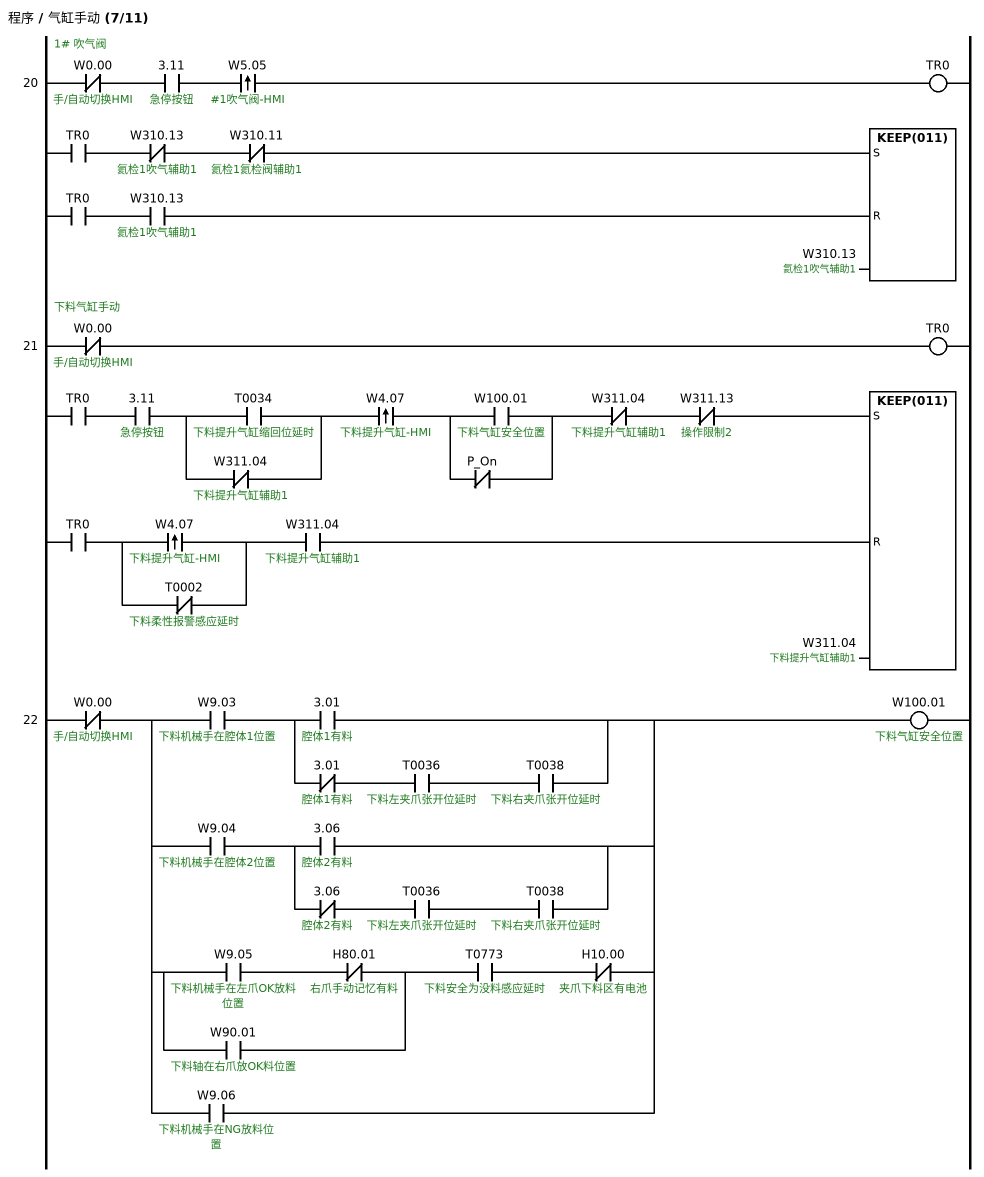
; [picture p120: 程序 / 气缸手动, rungs 20-22]
; rung 20: 1# 吹气阀
LDNOT W0.00  ; 手/自动切换HMI
AND 3.11  ; 急停按钮
@AND W5.05  ; #1吹气阀-HMI
OUT TR0
ANDNOT W310.13  ; 氦检1吹气辅助1
ANDNOT W310.11  ; 氦检1氦检阀辅助1
LD TR0
AND W310.13  ; 氦检1吹气辅助1
KEEP(011) W310.13  ; 氦检1吹气辅助1
; rung 21: 下料气缸手动
LDNOT W0.00  ; 手/自动切换HMI
OUT TR0
AND 3.11  ; 急停按钮
LD T0034  ; 下料提升气缸缩回位延时
ORNOT W311.04  ; 下料提升气缸辅助1
ANDLD
@AND W4.07  ; 下料提升气缸-HMI
LD W100.01  ; 下料气缸安全位置
ORNOT P_On
ANDLD
ANDNOT W311.04  ; 下料提升气缸辅助1
ANDNOT W311.13  ; 操作限制2
LD TR0
@LD W4.07  ; 下料提升气缸-HMI
ORNOT T0002  ; 下料柔性报警感应延时
ANDLD
AND W311.04  ; 下料提升气缸辅助1
KEEP(011) W311.04  ; 下料提升气缸辅助1
; rung 22
LDNOT W0.00  ; 手/自动切换HMI
LD W9.03  ; 下料机械手在腔体1位置
LD 3.01  ; 腔体1有料
LDNOT 3.01  ; 腔体1有料
AND T0036  ; 下料左夹爪张开位延时
AND T0038  ; 下料右夹爪张开位延时
ORLD
ANDLD
LD W9.04  ; 下料机械手在腔体2位置
LD 3.06  ; 腔体2有料
LDNOT 3.06  ; 腔体2有料
AND T0036  ; 下料左夹爪张开位延时
AND T0038  ; 下料右夹爪张开位延时
ORLD
ANDLD
ORLD
LD W9.05  ; 下料机械手在左爪OK放料位置
ANDNOT H80.01  ; 右爪手动记忆有料
OR W90.01  ; 下料轴在右爪放OK料位置
AND T0773  ; 下料安全为没料感应延时
ANDNOT H10.00  ; 夹爪下料区有电池
ORLD
OR W9.06  ; 下料机械手在NG放料位置
ANDLD
OUT W100.01  ; 下料气缸安全位置

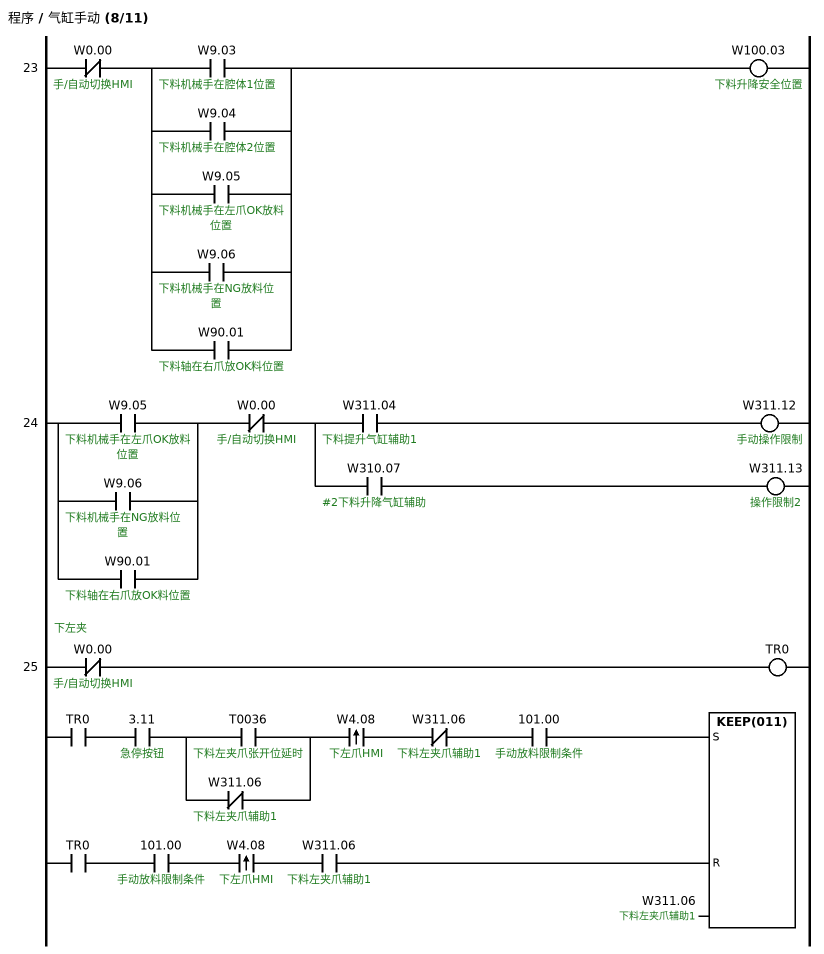
; rung 23
LDNOT W0.00  ; 手/自动切换HMI
LD W9.03  ; 下料机械手在腔体1位置
OR W9.04  ; 下料机械手在腔体2位置
OR W9.05  ; 下料机械手在左爪OK放料位置
OR W9.06  ; 下料机械手在NG放料位置
OR W90.01  ; 下料轴在右爪放OK料位置
ANDLD
OUT W100.03  ; 下料升降安全位置
; rung 24
LD W9.05  ; 下料机械手在左爪OK放料位置
OR W9.06  ; 下料机械手在NG放料位置
OR W90.01  ; 下料轴在右爪放OK料位置
ANDNOT W0.00  ; 手/自动切换HMI
OUT TR0
AND W311.04  ; 下料提升气缸辅助1
OUT W311.12  ; 手动操作限制
LD TR0
AND W310.07  ; #2下料升降气缸辅助
OUT W311.13  ; 操作限制2
; rung 25: 下左夹
LDNOT W0.00  ; 手/自动切换HMI
OUT TR0
AND 3.11  ; 急停按钮
LD T0036  ; 下料左夹爪张开位延时
ORNOT W311.06  ; 下料左夹爪辅助1
ANDLD
@AND W4.08  ; 下左爪HMI
ANDNOT W311.06  ; 下料左夹爪辅助1
AND 101.00  ; 手动放料限制条件
LD TR0
AND 101.00  ; 手动放料限制条件
@AND W4.08  ; 下左爪HMI
AND W311.06  ; 下料左夹爪辅助1
KEEP(011) W311.06  ; 下料左夹爪辅助1

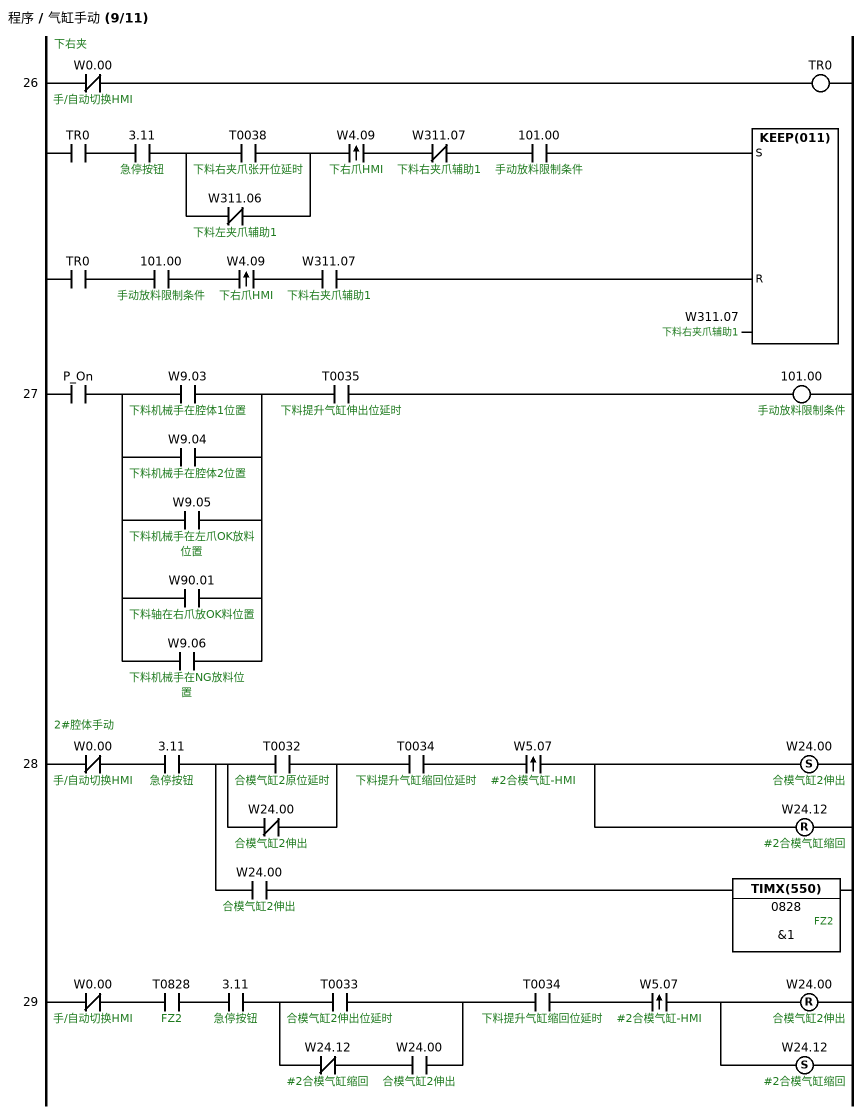
; rung 26: 下右夹
LDNOT W0.00  ; 手/自动切换HMI
OUT TR0
AND 3.11  ; 急停按钮
LD T0038  ; 下料右夹爪张开位延时
ORNOT W311.06  ; 下料左夹爪辅助1
ANDLD
@AND W4.09  ; 下右爪HMI
ANDNOT W311.07  ; 下料右夹爪辅助1
AND 101.00  ; 手动放料限制条件
LD TR0
AND 101.00  ; 手动放料限制条件
@AND W4.09  ; 下右爪HMI
AND W311.07  ; 下料右夹爪辅助1
KEEP(011) W311.07  ; 下料右夹爪辅助1
; rung 27
LD P_On
LD W9.03  ; 下料机械手在腔体1位置
OR W9.04  ; 下料机械手在腔体2位置
OR W9.05  ; 下料机械手在左爪OK放料位置
OR W90.01  ; 下料轴在右爪放OK料位置
OR W9.06  ; 下料机械手在NG放料位置
ANDLD
AND T0035  ; 下料提升气缸伸出位延时
OUT 101.00  ; 手动放料限制条件
; rung 28: 2#腔体手动
LDNOT W0.00  ; 手/自动切换HMI
AND 3.11  ; 急停按钮
OUT TR0
LD T0032  ; 合模气缸2原位延时
ORNOT W24.00  ; 合模气缸2伸出
ANDLD
AND T0034  ; 下料提升气缸缩回位延时
@AND W5.07  ; #2合模气缸-HMI
SET W24.00  ; 合模气缸2伸出
RSET W24.12  ; #2合模气缸缩回
LD TR0
AND W24.00  ; 合模气缸2伸出
TIMX(550) 0828 &1  ; FZ2
; rung 29
LDNOT W0.00  ; 手/自动切换HMI
AND T0828  ; FZ2
AND 3.11  ; 急停按钮
LD T0033  ; 合模气缸2伸出位延时
LDNOT W24.12  ; #2合模气缸缩回
AND W24.00  ; 合模气缸2伸出
ORLD
ANDLD
AND T0034  ; 下料提升气缸缩回位延时
@AND W5.07  ; #2合模气缸-HMI
RSET W24.00  ; 合模气缸2伸出
SET W24.12  ; #2合模气缸缩回

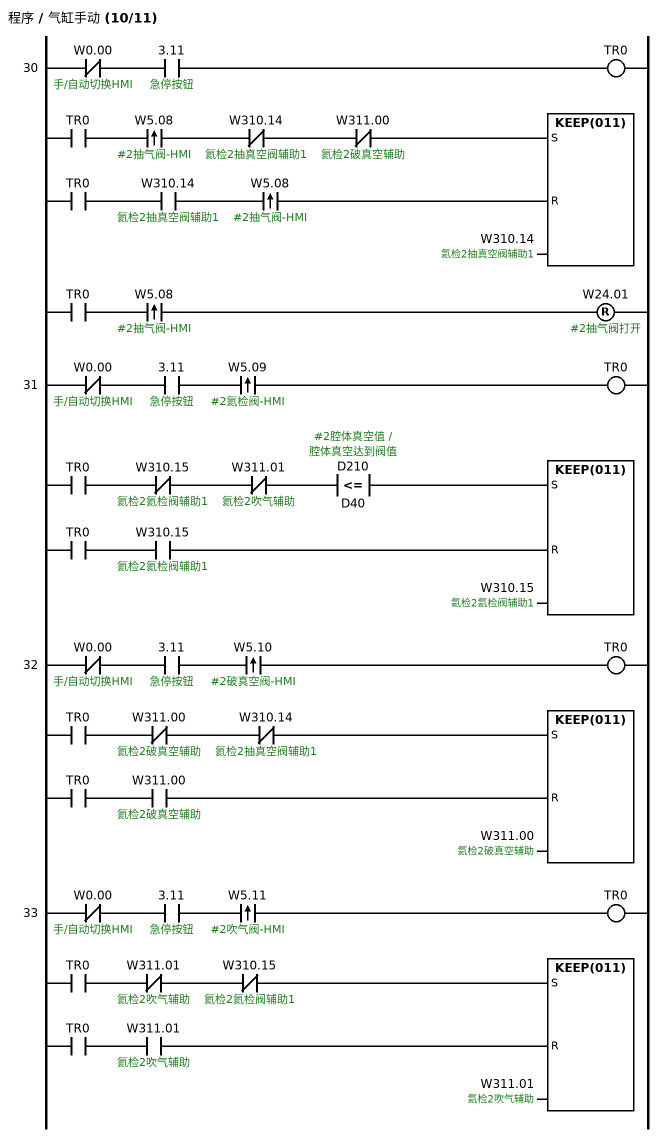
; rung 30
LDNOT W0.00  ; 手/自动切换HMI
AND 3.11  ; 急停按钮
OUT TR0
@AND W5.08  ; #2抽气阀-HMI
ANDNOT W310.14  ; 氦检2抽真空阀辅助1
ANDNOT W311.00  ; 氦检2破真空辅助
LD TR0
AND W310.14  ; 氦检2抽真空阀辅助1
@AND W5.08  ; #2抽气阀-HMI
KEEP(011) W310.14  ; 氦检2抽真空阀辅助1
LD TR0
@AND W5.08  ; #2抽气阀-HMI
RSET W24.01  ; #2抽气阀打开
; rung 31
LDNOT W0.00  ; 手/自动切换HMI
AND 3.11  ; 急停按钮
@AND W5.09  ; #2氦检阀-HMI
OUT TR0
ANDNOT W310.15  ; 氦检2氦检阀辅助1
ANDNOT W311.01  ; 氦检2吹气辅助
AND<=F(332) D210 D40  ; #2腔体真空值, 腔体真空达到阀值
LD TR0
AND W310.15  ; 氦检2氦检阀辅助1
KEEP(011) W310.15  ; 氦检2氦检阀辅助1
; rung 32
LDNOT W0.00  ; 手/自动切换HMI
AND 3.11  ; 急停按钮
@AND W5.10  ; #2破真空阀-HMI
OUT TR0
ANDNOT W311.00  ; 氦检2破真空辅助
ANDNOT W310.14  ; 氦检2抽真空阀辅助1
LD TR0
AND W311.00  ; 氦检2破真空辅助
KEEP(011) W311.00  ; 氦检2破真空辅助
; rung 33
LDNOT W0.00  ; 手/自动切换HMI
AND 3.11  ; 急停按钮
@AND W5.11  ; #2吹气阀-HMI
OUT TR0
ANDNOT W311.01  ; 氦检2吹气辅助
ANDNOT W310.15  ; 氦检2氦检阀辅助1
LD TR0
AND W311.01  ; 氦检2吹气辅助
KEEP(011) W311.01  ; 氦检2吹气辅助

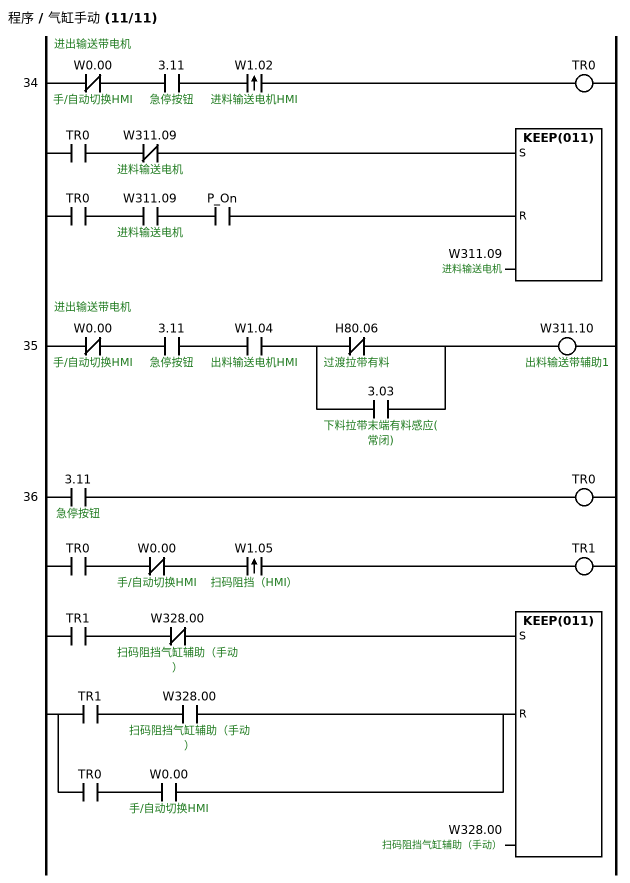
; rung 34: 进出输送带电机
LDNOT W0.00  ; 手/自动切换HMI
AND 3.11  ; 急停按钮
@AND W1.02  ; 进料输送电机HMI
OUT TR0
ANDNOT W311.09  ; 进料输送电机
LD TR0
AND W311.09  ; 进料输送电机
AND P_On
KEEP(011) W311.09  ; 进料输送电机
; rung 35: 进出输送带电机
LDNOT W0.00  ; 手/自动切换HMI
AND 3.11  ; 急停按钮
AND W1.04  ; 出料输送电机HMI
LDNOT H80.06  ; 过渡拉带有料
OR 3.03  ; 下料拉带末端有料感应(常闭)
ANDLD
OUT W311.10  ; 出料输送带辅助1
; rung 36
LD 3.11  ; 急停按钮
OUT TR0
ANDNOT W0.00  ; 手/自动切换HMI
@AND W1.05  ; 扫码阻挡（HMI）
OUT TR1
ANDNOT W328.00  ; 扫码阻挡气缸辅助（手动）
LD TR1
AND W328.00  ; 扫码阻挡气缸辅助（手动）
LD TR0
AND W0.00  ; 手/自动切换HMI
ORLD
KEEP(011) W328.00  ; 扫码阻挡气缸辅助（手动）

### Section 伺服参数

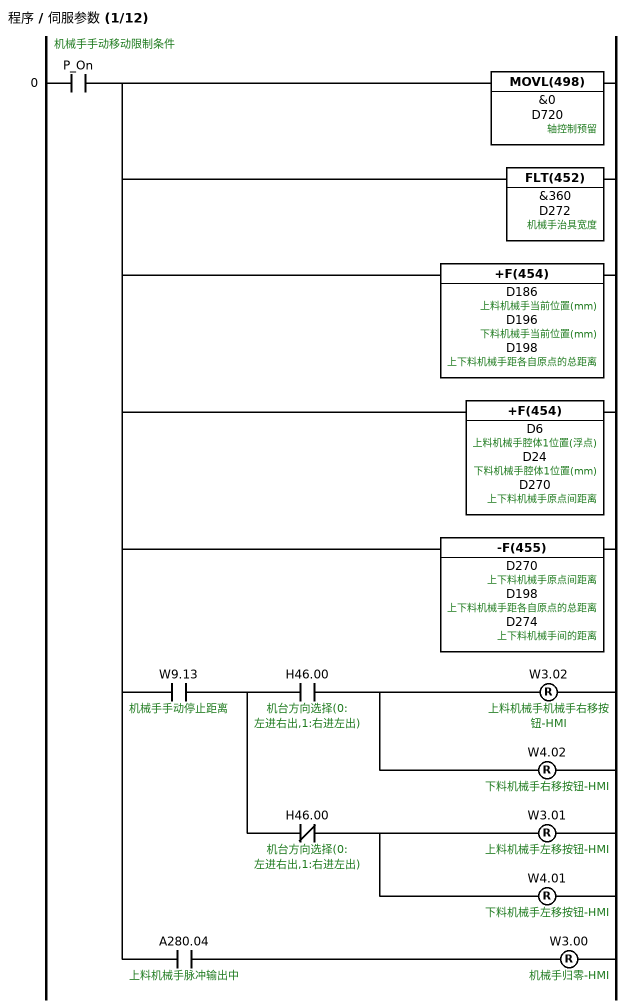
; rung 0: 机械手手动移动限制条件
LD P_On
OUT TR0
MOVL(498) &0 D720  ; 轴控制预留
FLT(452) &360 D272  ; 机械手治具宽度
+F(454) D186 D196 D198  ; 上料机械手当前位置(mm), 下料机械手当前位置(mm), 上下料机械手距各自原点的总距离
+F(454) D6 D24 D270  ; 上料机械手腔体1位置(浮点), 下料机械手腔体1位置(mm), 上下料机械手原点间距离
-F(455) D270 D198 D274  ; 上下料机械手原点间距离, 上下料机械手距各自原点的总距离, 上下料机械手间的距离
AND W9.13  ; 机械手手动停止距离
OUT TR1
AND H46.00  ; 机台方向选择(0:左进右出,1:右进左出)
RSET W3.02  ; 上料机械手机械手右移按钮-HMI
RSET W4.02  ; 下料机械手右移按钮-HMI
LD TR1
ANDNOT H46.00  ; 机台方向选择(0:左进右出,1:右进左出)
RSET W3.01  ; 上料机械手左移按钮-HMI
RSET W4.01  ; 下料机械手左移按钮-HMI
LD TR0
AND A280.04  ; 上料机械手脉冲输出中
RSET W3.00  ; 机械手归零-HMI

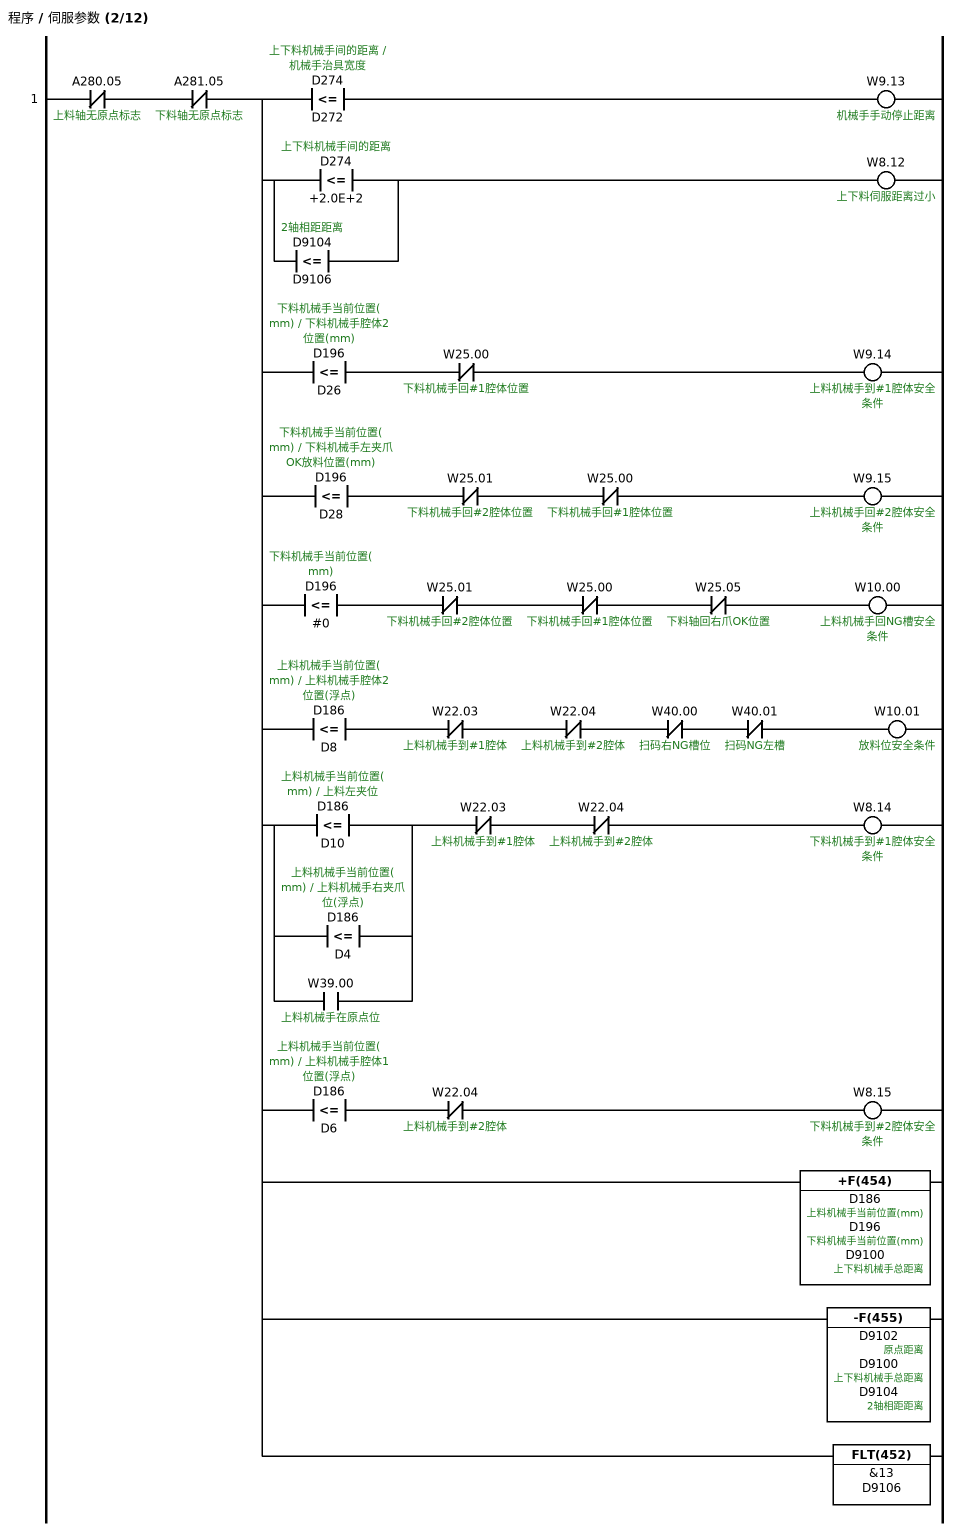
; rung 1
LDNOT A280.05  ; 上料轴无原点标志
ANDNOT A281.05  ; 下料轴无原点标志
OUT TR0
AND<=F(332) D274 D272  ; 上下料机械手间的距离, 机械手治具宽度
OUT W9.13  ; 机械手手动停止距离
LD TR0
LD<=F(332) D274 +2.0E+2  ; 上下料机械手间的距离
OR<=F(332) D9104 D9106  ; 2轴相距距离
ANDLD
OUT W8.12  ; 上下料伺服距离过小
LD TR0
AND<=F(332) D196 D26  ; 下料机械手当前位置(mm), 下料机械手腔体2位置(mm)
ANDNOT W25.00  ; 下料机械手回#1腔体位置
OUT W9.14  ; 上料机械手到#1腔体安全条件
LD TR0
AND<=F(332) D196 D28  ; 下料机械手当前位置(mm), 下料机械手左夹爪OK放料位置(mm)
ANDNOT W25.01  ; 下料机械手回#2腔体位置
ANDNOT W25.00  ; 下料机械手回#1腔体位置
OUT W9.15  ; 上料机械手回#2腔体安全条件
LD TR0
AND<=F(332) D196 #0  ; 下料机械手当前位置(mm)
ANDNOT W25.01  ; 下料机械手回#2腔体位置
ANDNOT W25.00  ; 下料机械手回#1腔体位置
ANDNOT W25.05  ; 下料轴回右爪OK位置
OUT W10.00  ; 上料机械手回NG槽安全条件
LD TR0
AND<=F(332) D186 D8  ; 上料机械手当前位置(mm), 上料机械手腔体2位置(浮点)
ANDNOT W22.03  ; 上料机械手到#1腔体
ANDNOT W22.04  ; 上料机械手到#2腔体
ANDNOT W40.00  ; 扫码右NG槽位
ANDNOT W40.01  ; 扫码NG左槽
OUT W10.01  ; 放料位安全条件
LD TR0
LD<=F(332) D186 D10  ; 上料机械手当前位置(mm), 上料左夹位
OR<=F(332) D186 D4  ; 上料机械手当前位置(mm), 上料机械手右夹爪位(浮点)
OR W39.00  ; 上料机械手在原点位
ANDLD
ANDNOT W22.03  ; 上料机械手到#1腔体
ANDNOT W22.04  ; 上料机械手到#2腔体
OUT W8.14  ; 下料机械手到#1腔体安全条件
LD TR0
AND<=F(332) D186 D6  ; 上料机械手当前位置(mm), 上料机械手腔体1位置(浮点)
ANDNOT W22.04  ; 上料机械手到#2腔体
OUT W8.15  ; 下料机械手到#2腔体安全条件
LD TR0
+F(454) D186 D196 D9100  ; 上料机械手当前位置(mm), 下料机械手当前位置(mm), 上下料机械手总距离
-F(455) D9102 D9100 D9104  ; 原点距离, 上下料机械手总距离, 2轴相距距离
FLT(452) &13 D9106

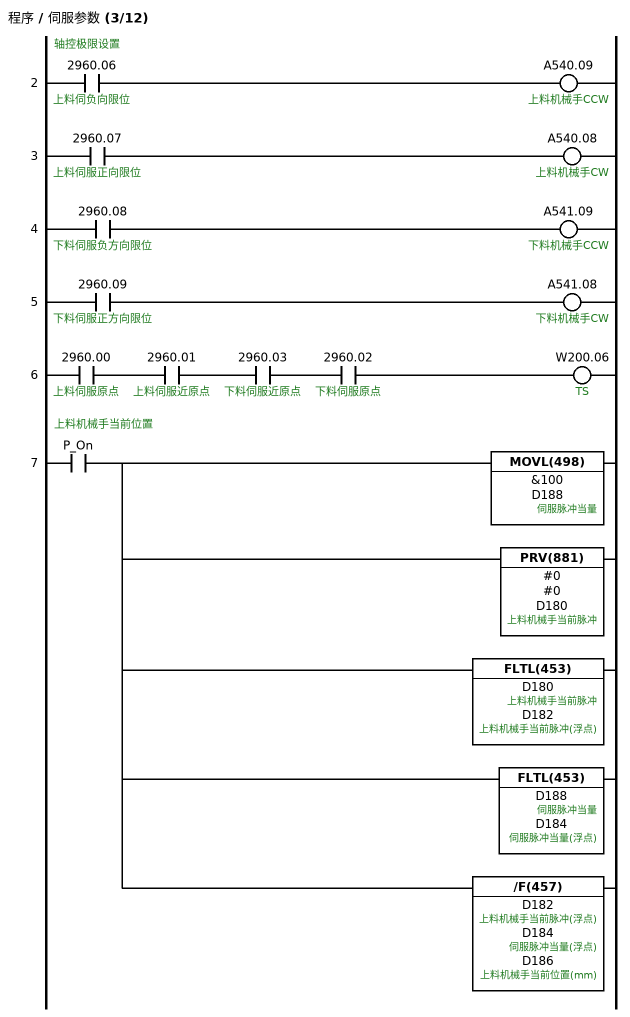
; rung 2: 轴控极限设置
LD 2960.06  ; 上料伺负向限位
OUT A540.09  ; 上料机械手CCW
; rung 3
LD 2960.07  ; 上料伺服正向限位
OUT A540.08  ; 上料机械手CW
; rung 4
LD 2960.08  ; 下料伺服负方向限位
OUT A541.09  ; 下料机械手CCW
; rung 5
LD 2960.09  ; 下料伺服正方向限位
OUT A541.08  ; 下料机械手CW
; rung 6
LD 2960.00  ; 上料伺服原点
AND 2960.01  ; 上料伺服近原点
AND 2960.03  ; 下料伺服近原点
AND 2960.02  ; 下料伺服原点
OUT W200.06  ; TS
; rung 7: 上料机械手当前位置
LD P_On
MOVL(498) &100 D188  ; 伺服脉冲当量
PRV(881) #0 #0 D180  ; 上料机械手当前脉冲
FLTL(453) D180 D182  ; 上料机械手当前脉冲, 上料机械手当前脉冲(浮点)
FLTL(453) D188 D184  ; 伺服脉冲当量, 伺服脉冲当量(浮点)
/F(457) D182 D184 D186  ; 上料机械手当前脉冲(浮点), 伺服脉冲当量(浮点), 上料机械手当前位置(mm)

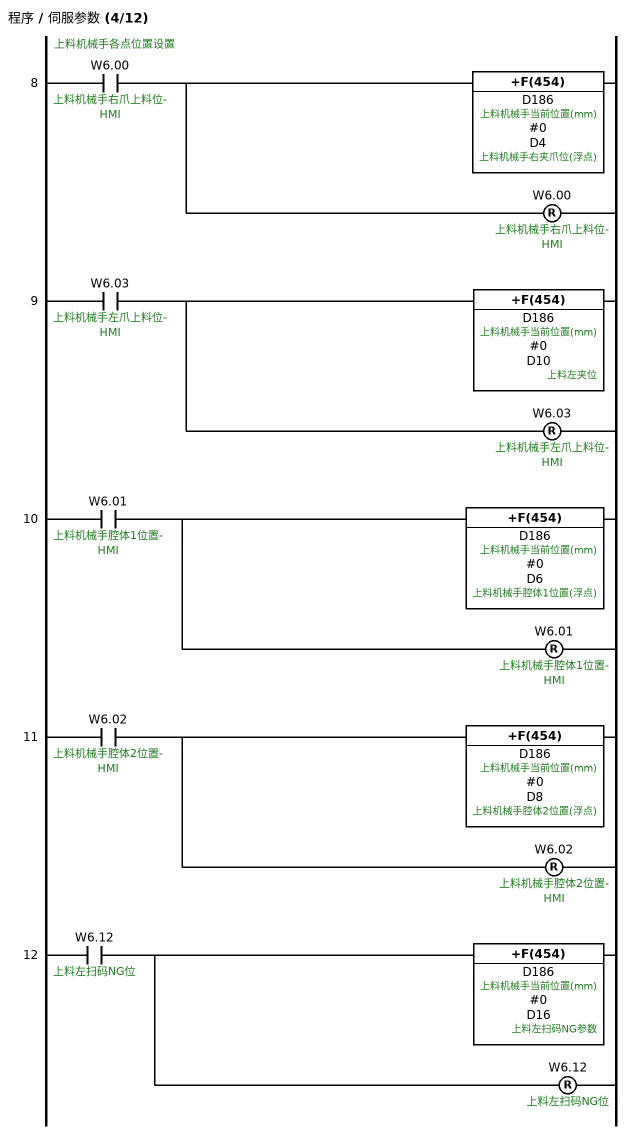
; rung 8: 上料机械手各点位置设置
LD W6.00  ; 上料机械手右爪上料位-HMI
+F(454) D186 #0 D4  ; 上料机械手当前位置(mm), 上料机械手右夹爪位(浮点)
RSET W6.00  ; 上料机械手右爪上料位-HMI
; rung 9
LD W6.03  ; 上料机械手左爪上料位-HMI
+F(454) D186 #0 D10  ; 上料机械手当前位置(mm), 上料左夹位
RSET W6.03  ; 上料机械手左爪上料位-HMI
; rung 10
LD W6.01  ; 上料机械手腔体1位置-HMI
+F(454) D186 #0 D6  ; 上料机械手当前位置(mm), 上料机械手腔体1位置(浮点)
RSET W6.01  ; 上料机械手腔体1位置-HMI
; rung 11
LD W6.02  ; 上料机械手腔体2位置-HMI
+F(454) D186 #0 D8  ; 上料机械手当前位置(mm), 上料机械手腔体2位置(浮点)
RSET W6.02  ; 上料机械手腔体2位置-HMI
; rung 12
LD W6.12  ; 上料左扫码NG位
+F(454) D186 #0 D16  ; 上料机械手当前位置(mm), 上料左扫码NG参数
RSET W6.12  ; 上料左扫码NG位

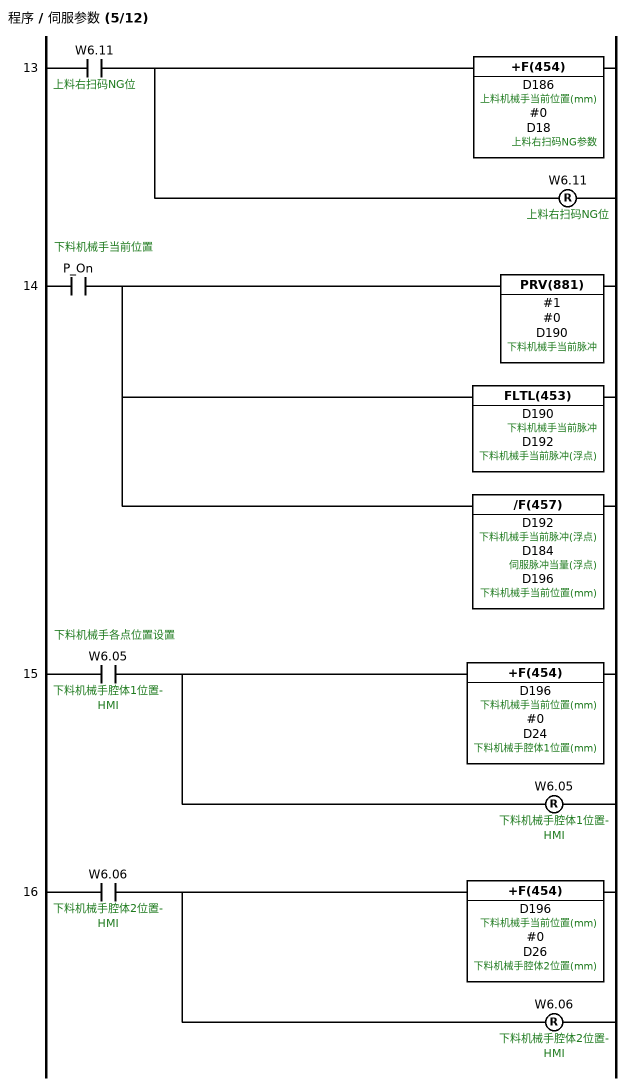
; rung 13
LD W6.11  ; 上料右扫码NG位
+F(454) D186 #0 D18  ; 上料机械手当前位置(mm), 上料右扫码NG参数
RSET W6.11  ; 上料右扫码NG位
; rung 14: 下料机械手当前位置
LD P_On
PRV(881) #1 #0 D190  ; 下料机械手当前脉冲
FLTL(453) D190 D192  ; 下料机械手当前脉冲, 下料机械手当前脉冲(浮点)
/F(457) D192 D184 D196  ; 下料机械手当前脉冲(浮点), 伺服脉冲当量(浮点), 下料机械手当前位置(mm)
; rung 15: 下料机械手各点位置设置
LD W6.05  ; 下料机械手腔体1位置-HMI
+F(454) D196 #0 D24  ; 下料机械手当前位置(mm), 下料机械手腔体1位置(mm)
RSET W6.05  ; 下料机械手腔体1位置-HMI
; rung 16
LD W6.06  ; 下料机械手腔体2位置-HMI
+F(454) D196 #0 D26  ; 下料机械手当前位置(mm), 下料机械手腔体2位置(mm)
RSET W6.06  ; 下料机械手腔体2位置-HMI

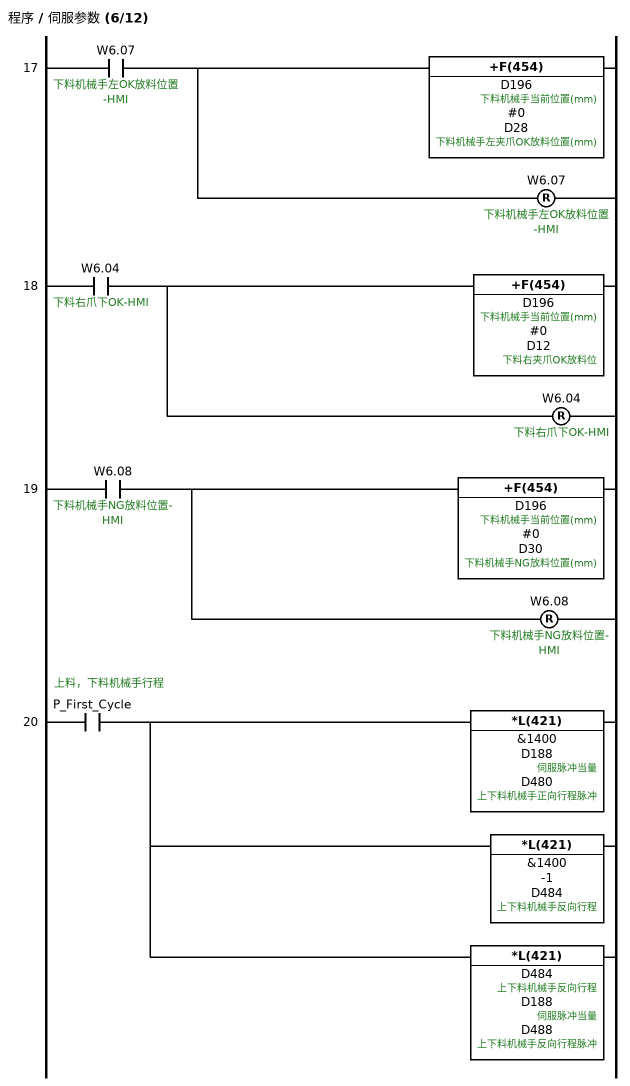
; rung 17
LD W6.07  ; 下料机械手左OK放料位置-HMI
+F(454) D196 #0 D28  ; 下料机械手当前位置(mm), 下料机械手左夹爪OK放料位置(mm)
RSET W6.07  ; 下料机械手左OK放料位置-HMI
; rung 18
LD W6.04  ; 下料右爪下OK-HMI
+F(454) D196 #0 D12  ; 下料机械手当前位置(mm), 下料右夹爪OK放料位
RSET W6.04  ; 下料右爪下OK-HMI
; rung 19
LD W6.08  ; 下料机械手NG放料位置-HMI
+F(454) D196 #0 D30  ; 下料机械手当前位置(mm), 下料机械手NG放料位置(mm)
RSET W6.08  ; 下料机械手NG放料位置-HMI
; rung 20: 上料，下料机械手行程
LD P_First_Cycle
*L(421) &1400 D188 D480  ; 伺服脉冲当量, 上下料机械手正向行程脉冲
*L(421) &1400 -1 D484  ; 上下料机械手反向行程
*L(421) D484 D188 D488  ; 上下料机械手反向行程, 伺服脉冲当量, 上下料机械手反向行程脉冲

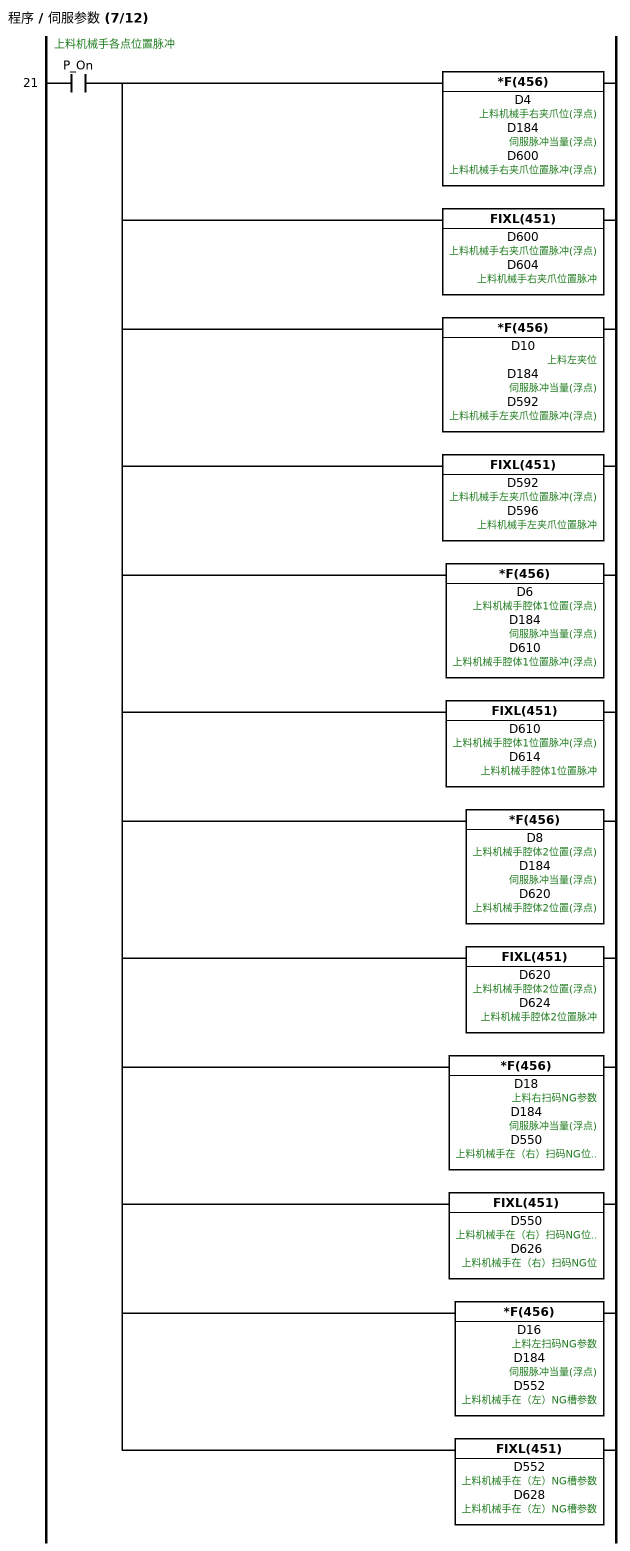
; rung 21: 上料机械手各点位置脉冲
LD P_On
*F(456) D4 D184 D600  ; 上料机械手右夹爪位(浮点), 伺服脉冲当量(浮点), 上料机械手右夹爪位置脉冲(浮点)
FIXL(451) D600 D604  ; 上料机械手右夹爪位置脉冲(浮点), 上料机械手右夹爪位置脉冲
*F(456) D10 D184 D592  ; 上料左夹位, 伺服脉冲当量(浮点), 上料机械手左夹爪位置脉冲(浮点)
FIXL(451) D592 D596  ; 上料机械手左夹爪位置脉冲(浮点), 上料机械手左夹爪位置脉冲
*F(456) D6 D184 D610  ; 上料机械手腔体1位置(浮点), 伺服脉冲当量(浮点), 上料机械手腔体1位置脉冲(浮点)
FIXL(451) D610 D614  ; 上料机械手腔体1位置脉冲(浮点), 上料机械手腔体1位置脉冲
*F(456) D8 D184 D620  ; 上料机械手腔体2位置(浮点), 伺服脉冲当量(浮点)
FIXL(451) D620 D624  ; 上料机械手腔体2位置(浮点), 上料机械手腔体2位置脉冲
*F(456) D18 D184 D550  ; 上料右扫码NG参数, 伺服脉冲当量(浮点), 上料机械手在（右）扫码NG位..
FIXL(451) D550 D626  ; 上料机械手在（右）扫码NG位.., 上料机械手在（右）扫码NG位
*F(456) D16 D184 D552  ; 上料左扫码NG参数, 伺服脉冲当量(浮点), 上料机械手在（左）NG槽参数
FIXL(451) D552 D628  ; 上料机械手在（左）NG槽参数

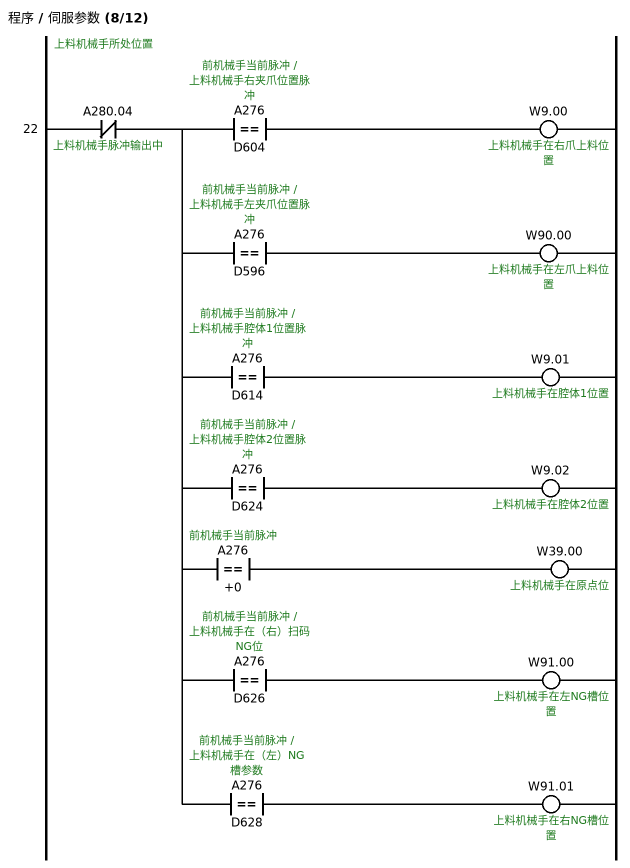
; rung 22: 上料机械手所处位置
LDNOT A280.04  ; 上料机械手脉冲输出中
OUT TR0
AND=SL(303) A276 D604  ; 前机械手当前脉冲, 上料机械手右夹爪位置脉冲
OUT W9.00  ; 上料机械手在右爪上料位置
LD TR0
AND=SL(303) A276 D596  ; 前机械手当前脉冲, 上料机械手左夹爪位置脉冲
OUT W90.00  ; 上料机械手在左爪上料位置
LD TR0
AND=SL(303) A276 D614  ; 前机械手当前脉冲, 上料机械手腔体1位置脉冲
OUT W9.01  ; 上料机械手在腔体1位置
LD TR0
AND=SL(303) A276 D624  ; 前机械手当前脉冲, 上料机械手腔体2位置脉冲
OUT W9.02  ; 上料机械手在腔体2位置
LD TR0
AND=SL(303) A276 +0  ; 前机械手当前脉冲
OUT W39.00  ; 上料机械手在原点位
LD TR0
AND=SL(303) A276 D626  ; 前机械手当前脉冲, 上料机械手在（右）扫码NG位
OUT W91.00  ; 上料机械手在左NG槽位置
LD TR0
AND=SL(303) A276 D628  ; 前机械手当前脉冲, 上料机械手在（左）NG槽参数
OUT W91.01  ; 上料机械手在右NG槽位置

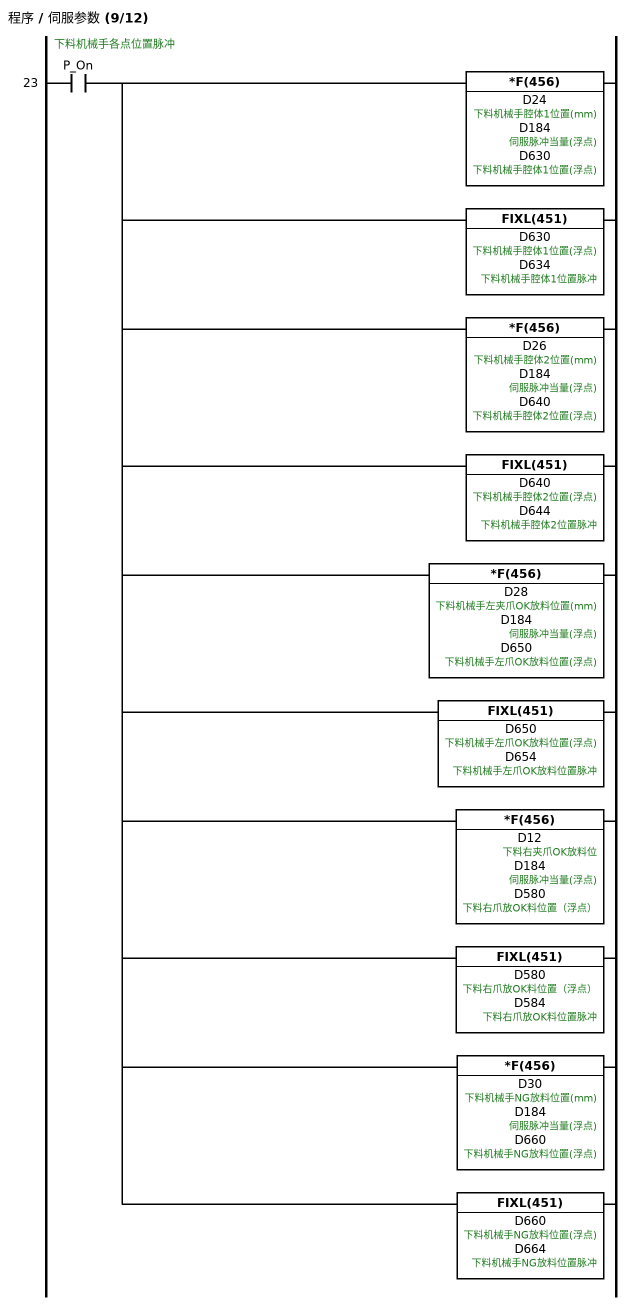
; rung 23: 下料机械手各点位置脉冲
LD P_On
*F(456) D24 D184 D630  ; 下料机械手腔体1位置(mm), 伺服脉冲当量(浮点), 下料机械手腔体1位置(浮点)
FIXL(451) D630 D634  ; 下料机械手腔体1位置(浮点), 下料机械手腔体1位置脉冲
*F(456) D26 D184 D640  ; 下料机械手腔体2位置(mm), 伺服脉冲当量(浮点), 下料机械手腔体2位置(浮点)
FIXL(451) D640 D644  ; 下料机械手腔体2位置(浮点), 下料机械手腔体2位置脉冲
*F(456) D28 D184 D650  ; 下料机械手左夹爪OK放料位置(mm), 伺服脉冲当量(浮点), 下料机械手左爪OK放料位置(浮点)
FIXL(451) D650 D654  ; 下料机械手左爪OK放料位置(浮点), 下料机械手左爪OK放料位置脉冲
*F(456) D12 D184 D580  ; 下料右夹爪OK放料位, 伺服脉冲当量(浮点), 下料右爪放OK料位置（浮点）
FIXL(451) D580 D584  ; 下料右爪放OK料位置（浮点）, 下料右爪放OK料位置脉冲
*F(456) D30 D184 D660  ; 下料机械手NG放料位置(mm), 伺服脉冲当量(浮点), 下料机械手NG放料位置(浮点)
FIXL(451) D660 D664  ; 下料机械手NG放料位置(浮点), 下料机械手NG放料位置脉冲

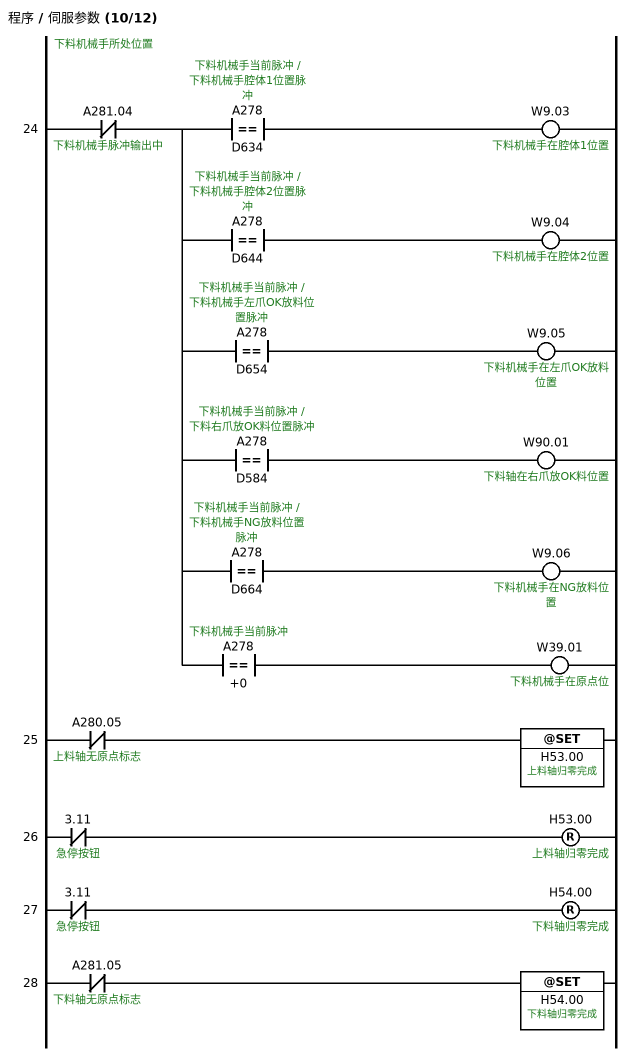
; rung 24: 下料机械手所处位置
LDNOT A281.04  ; 下料机械手脉冲输出中
OUT TR0
AND=SL(303) A278 D634  ; 下料机械手当前脉冲, 下料机械手腔体1位置脉冲
OUT W9.03  ; 下料机械手在腔体1位置
LD TR0
AND=SL(303) A278 D644  ; 下料机械手当前脉冲, 下料机械手腔体2位置脉冲
OUT W9.04  ; 下料机械手在腔体2位置
LD TR0
AND=SL(303) A278 D654  ; 下料机械手当前脉冲, 下料机械手左爪OK放料位置脉冲
OUT W9.05  ; 下料机械手在左爪OK放料位置
LD TR0
AND=SL(303) A278 D584  ; 下料机械手当前脉冲, 下料右爪放OK料位置脉冲
OUT W90.01  ; 下料轴在右爪放OK料位置
LD TR0
AND=SL(303) A278 D664  ; 下料机械手当前脉冲, 下料机械手NG放料位置脉冲
OUT W9.06  ; 下料机械手在NG放料位置
LD TR0
AND=SL(303) A278 +0  ; 下料机械手当前脉冲
OUT W39.01  ; 下料机械手在原点位
; rung 25
LDNOT A280.05  ; 上料轴无原点标志
@SET H53.00  ; 上料轴归零完成
; rung 26
LDNOT 3.11  ; 急停按钮
RSET H53.00  ; 上料轴归零完成
; rung 27
LDNOT 3.11  ; 急停按钮
RSET H54.00  ; 下料轴归零完成
; rung 28
LDNOT A281.05  ; 下料轴无原点标志
@SET H54.00  ; 下料轴归零完成

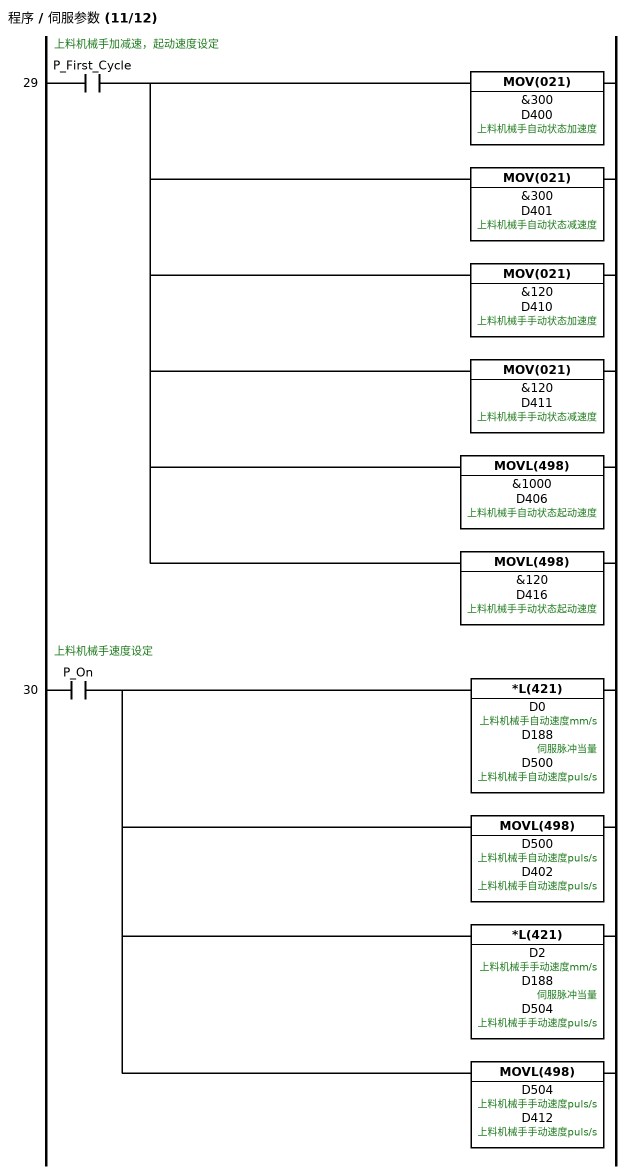
; rung 29: 上料机械手加减速，起动速度设定
LD P_First_Cycle
MOV(021) &300 D400  ; 上料机械手自动状态加速度
MOV(021) &300 D401  ; 上料机械手自动状态减速度
MOV(021) &120 D410  ; 上料机械手手动状态加速度
MOV(021) &120 D411  ; 上料机械手手动状态减速度
MOVL(498) &1000 D406  ; 上料机械手自动状态起动速度
MOVL(498) &120 D416  ; 上料机械手手动状态起动速度
; rung 30: 上料机械手速度设定
LD P_On
*L(421) D0 D188 D500  ; 上料机械手自动速度mm/s, 伺服脉冲当量, 上料机械手自动速度puls/s
MOVL(498) D500 D402  ; 上料机械手自动速度puls/s
*L(421) D2 D188 D504  ; 上料机械手手动速度mm/s, 伺服脉冲当量, 上料机械手手动速度puls/s
MOVL(498) D504 D412  ; 上料机械手手动速度puls/s

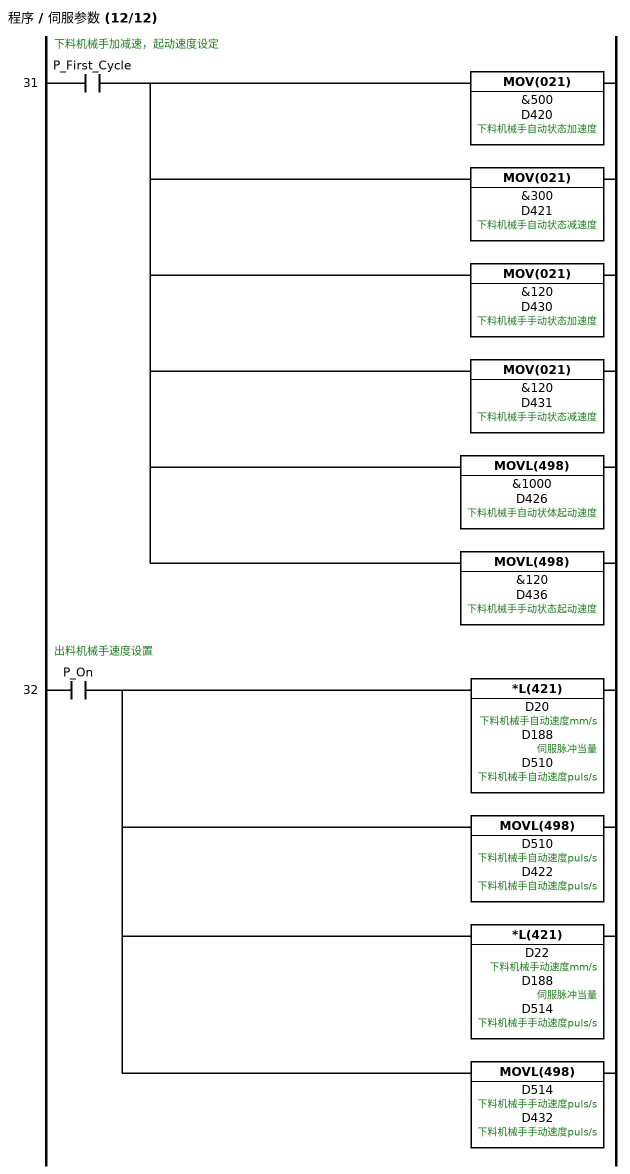
; rung 31: 下料机械手加减速，起动速度设定
LD P_First_Cycle
MOV(021) &500 D420  ; 下料机械手自动状态加速度
MOV(021) &300 D421  ; 下料机械手自动状态减速度
MOV(021) &120 D430  ; 下料机械手手动状态加速度
MOV(021) &120 D431  ; 下料机械手手动状态减速度
MOVL(498) &1000 D426  ; 下料机械手自动状体起动速度
MOVL(498) &120 D436  ; 下料机械手手动状态起动速度
; rung 32: 出料机械手速度设置
LD P_On
*L(421) D20 D188 D510  ; 下料机械手自动速度mm/s, 伺服脉冲当量, 下料机械手自动速度puls/s
MOVL(498) D510 D422  ; 下料机械手自动速度puls/s
*L(421) D22 D188 D514  ; 下料机械手动速度mm/s, 伺服脉冲当量, 下料机械手手动速度puls/s
MOVL(498) D514 D432  ; 下料机械手手动速度puls/s

### Section 伺服手动

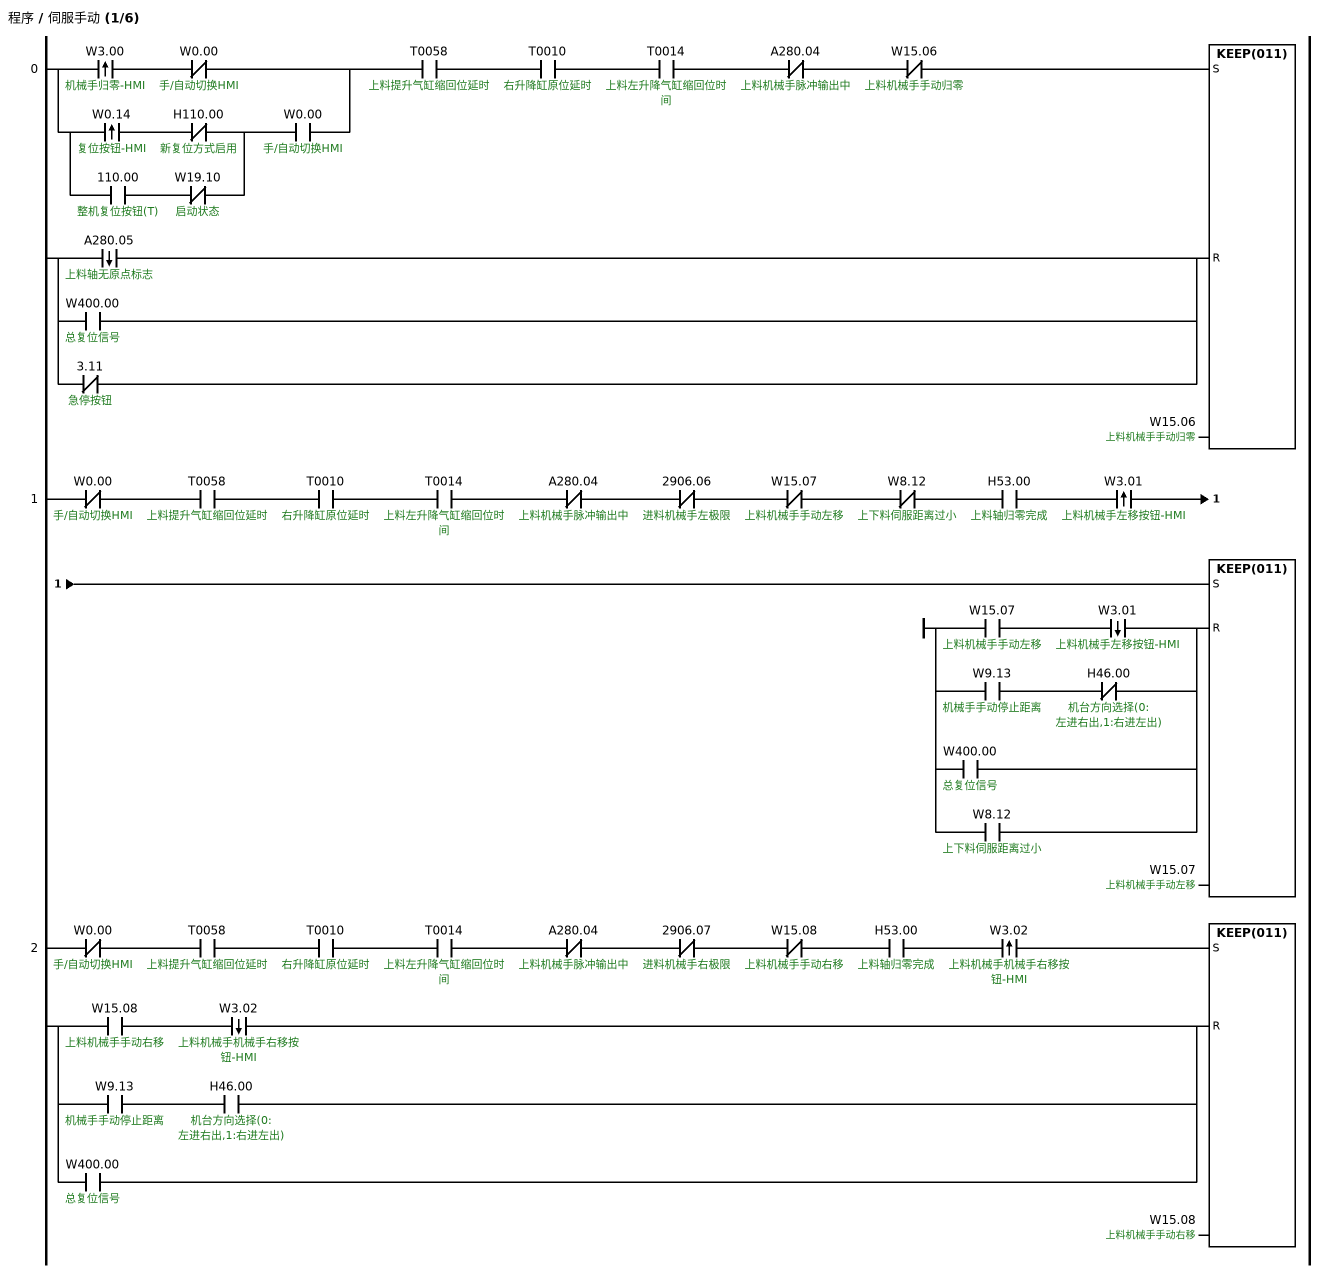
; rung 0
@LD W3.00  ; 机械手归零-HMI
ANDNOT W0.00  ; 手/自动切换HMI
@LD W0.14  ; 复位按钮-HMI
ANDNOT H110.00  ; 新复位方式启用
LD 110.00  ; 整机复位按钮(T)
ANDNOT W19.10  ; 启动状态
ORLD
AND W0.00  ; 手/自动切换HMI
ORLD
AND T0058  ; 上料提升气缸缩回位延时
AND T0010  ; 右升降缸原位延时
AND T0014  ; 上料左升降气缸缩回位时间
ANDNOT A280.04  ; 上料机械手脉冲输出中
ANDNOT W15.06  ; 上料机械手手动归零
%LD A280.05  ; 上料轴无原点标志
OR W400.00  ; 总复位信号
ORNOT 3.11  ; 急停按钮
KEEP(011) W15.06  ; 上料机械手手动归零
; rung 1
LDNOT W0.00  ; 手/自动切换HMI
AND T0058  ; 上料提升气缸缩回位延时
AND T0010  ; 右升降缸原位延时
AND T0014  ; 上料左升降气缸缩回位时间
ANDNOT A280.04  ; 上料机械手脉冲输出中
ANDNOT 2906.06  ; 进料机械手左极限
ANDNOT W15.07  ; 上料机械手手动左移
ANDNOT W8.12  ; 上下料伺服距离过小
AND H53.00  ; 上料轴归零完成
@AND W3.01  ; 上料机械手左移按钮-HMI
LD W15.07  ; 上料机械手手动左移
%AND W3.01  ; 上料机械手左移按钮-HMI
LD W9.13  ; 机械手手动停止距离
ANDNOT H46.00  ; 机台方向选择(0:左进右出,1:右进左出)
ORLD
OR W400.00  ; 总复位信号
OR W8.12  ; 上下料伺服距离过小
KEEP(011) W15.07  ; 上料机械手手动左移
; rung 2
LDNOT W0.00  ; 手/自动切换HMI
AND T0058  ; 上料提升气缸缩回位延时
AND T0010  ; 右升降缸原位延时
AND T0014  ; 上料左升降气缸缩回位时间
ANDNOT A280.04  ; 上料机械手脉冲输出中
ANDNOT 2906.07  ; 进料机械手右极限
ANDNOT W15.08  ; 上料机械手手动右移
AND H53.00  ; 上料轴归零完成
@AND W3.02  ; 上料机械手机械手右移按钮-HMI
LD W15.08  ; 上料机械手手动右移
%AND W3.02  ; 上料机械手机械手右移按钮-HMI
LD W9.13  ; 机械手手动停止距离
AND H46.00  ; 机台方向选择(0:左进右出,1:右进左出)
ORLD
OR W400.00  ; 总复位信号
KEEP(011) W15.08  ; 上料机械手手动右移

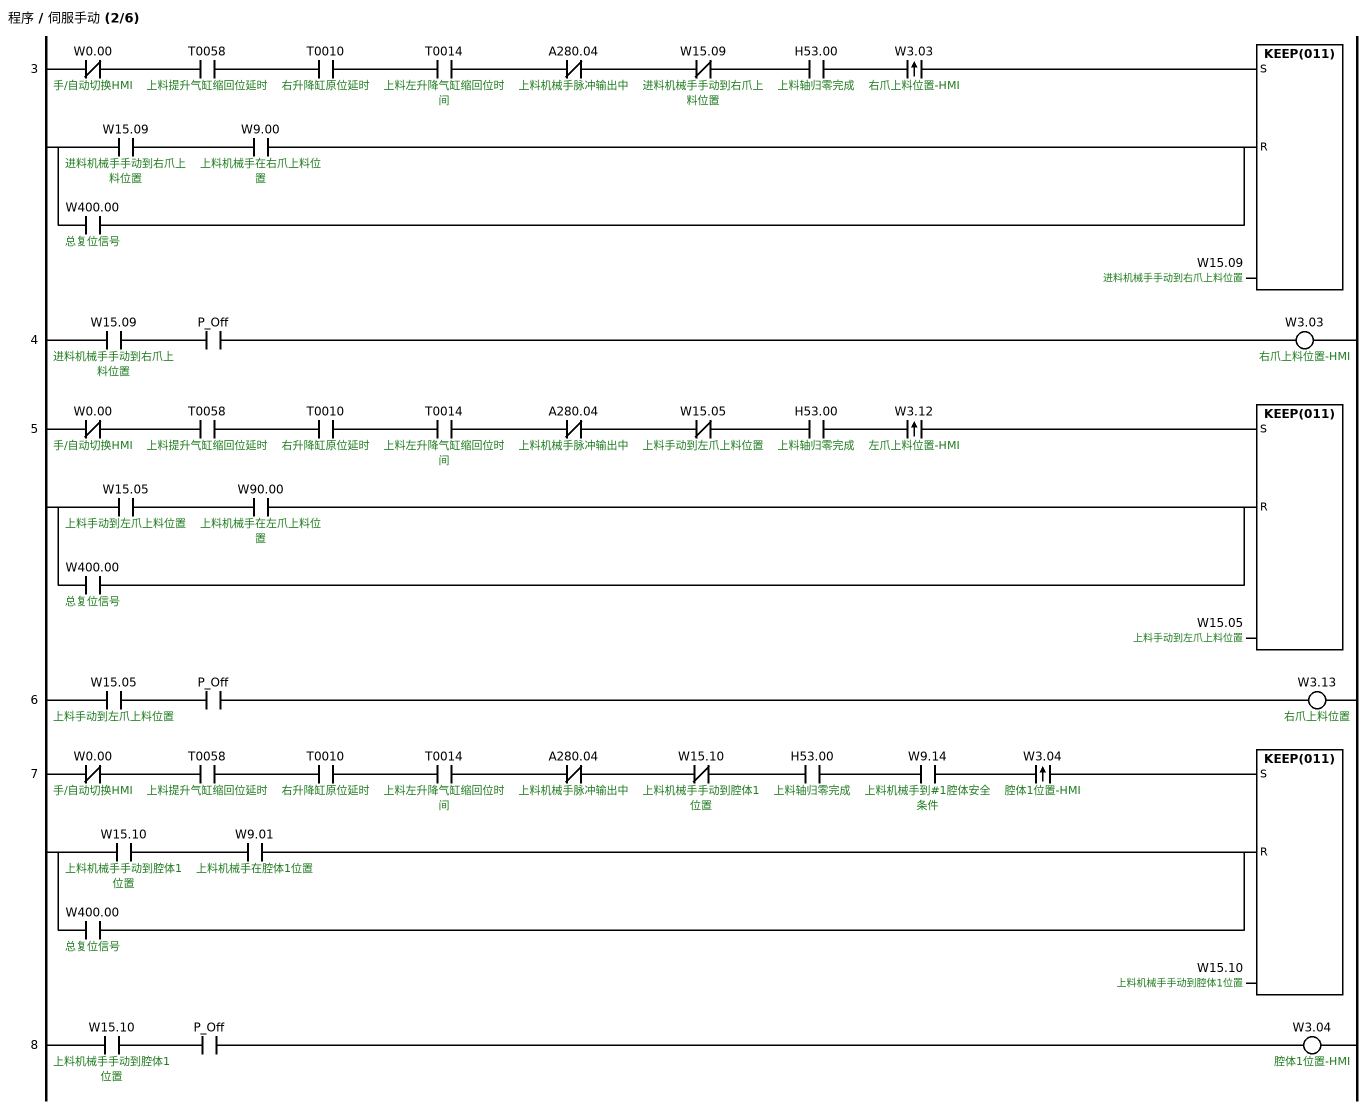
; rung 3
LDNOT W0.00  ; 手/自动切换HMI
AND T0058  ; 上料提升气缸缩回位延时
AND T0010  ; 右升降缸原位延时
AND T0014  ; 上料左升降气缸缩回位时间
ANDNOT A280.04  ; 上料机械手脉冲输出中
ANDNOT W15.09  ; 进料机械手手动到右爪上料位置
AND H53.00  ; 上料轴归零完成
@AND W3.03  ; 右爪上料位置-HMI
LD W15.09  ; 进料机械手手动到右爪上料位置
AND W9.00  ; 上料机械手在右爪上料位置
OR W400.00  ; 总复位信号
KEEP(011) W15.09  ; 进料机械手手动到右爪上料位置
; rung 4
LD W15.09  ; 进料机械手手动到右爪上料位置
AND P_Off
OUT W3.03  ; 右爪上料位置-HMI
; rung 5
LDNOT W0.00  ; 手/自动切换HMI
AND T0058  ; 上料提升气缸缩回位延时
AND T0010  ; 右升降缸原位延时
AND T0014  ; 上料左升降气缸缩回位时间
ANDNOT A280.04  ; 上料机械手脉冲输出中
ANDNOT W15.05  ; 上料手动到左爪上料位置
AND H53.00  ; 上料轴归零完成
@AND W3.12  ; 左爪上料位置-HMI
LD W15.05  ; 上料手动到左爪上料位置
AND W90.00  ; 上料机械手在左爪上料位置
OR W400.00  ; 总复位信号
KEEP(011) W15.05  ; 上料手动到左爪上料位置
; rung 6
LD W15.05  ; 上料手动到左爪上料位置
AND P_Off
OUT W3.13  ; 右爪上料位置
; rung 7
LDNOT W0.00  ; 手/自动切换HMI
AND T0058  ; 上料提升气缸缩回位延时
AND T0010  ; 右升降缸原位延时
AND T0014  ; 上料左升降气缸缩回位时间
ANDNOT A280.04  ; 上料机械手脉冲输出中
ANDNOT W15.10  ; 上料机械手手动到腔体1位置
AND H53.00  ; 上料轴归零完成
AND W9.14  ; 上料机械手到#1腔体安全条件
@AND W3.04  ; 腔体1位置-HMI
LD W15.10  ; 上料机械手手动到腔体1位置
AND W9.01  ; 上料机械手在腔体1位置
OR W400.00  ; 总复位信号
KEEP(011) W15.10  ; 上料机械手手动到腔体1位置
; rung 8
LD W15.10  ; 上料机械手手动到腔体1位置
AND P_Off
OUT W3.04  ; 腔体1位置-HMI

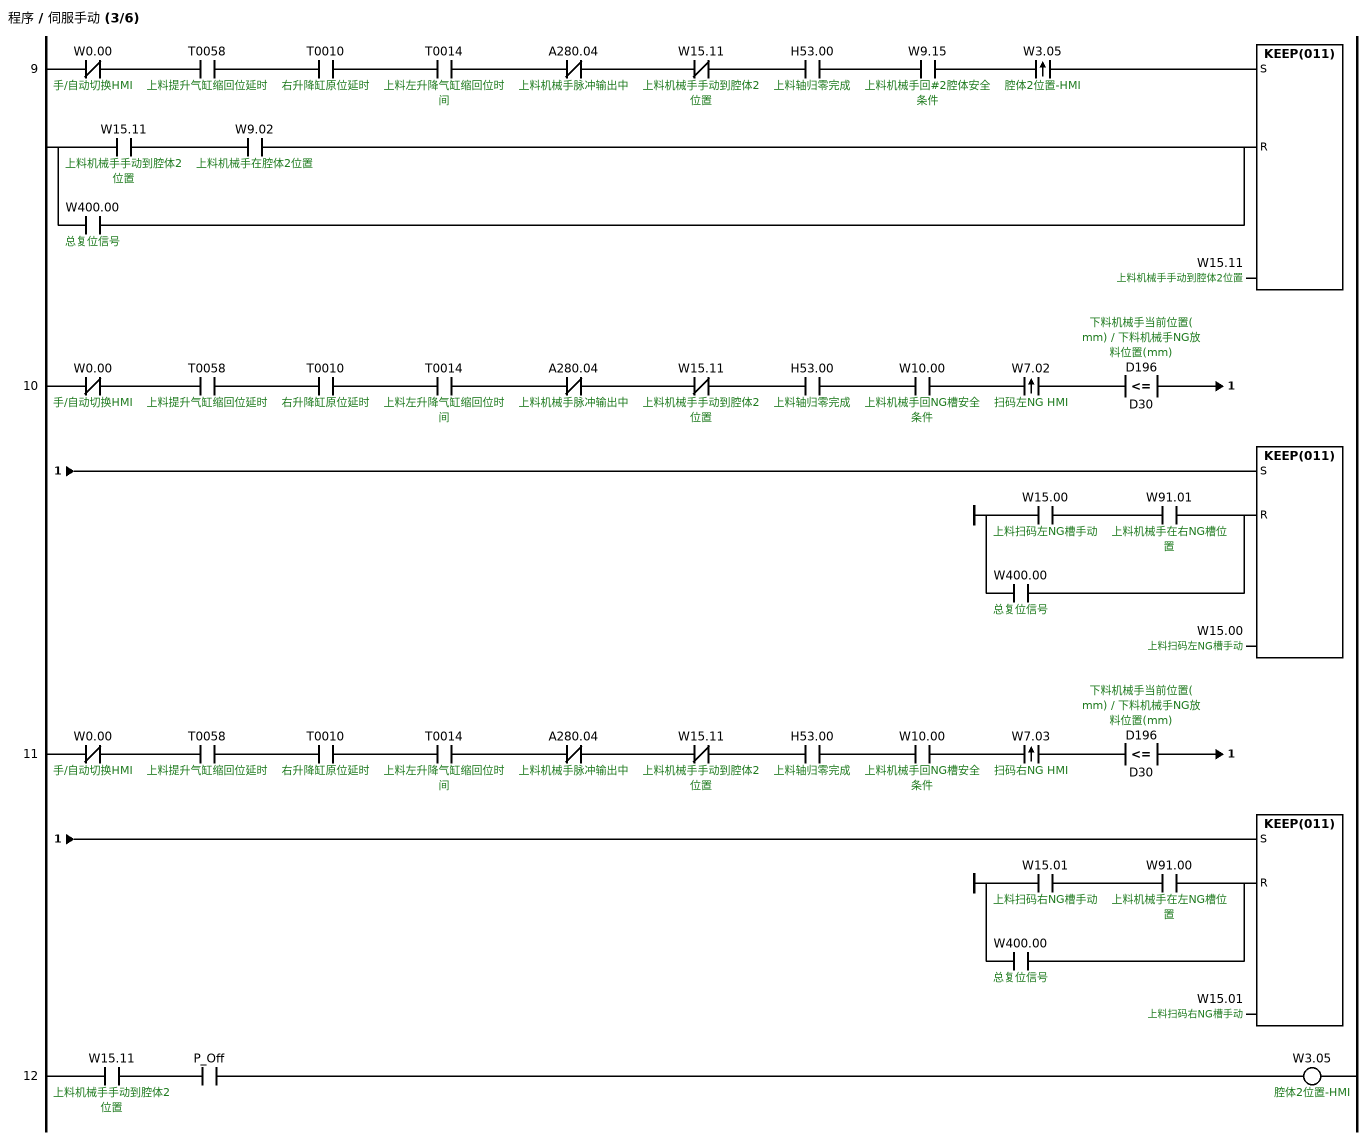
; rung 9
LDNOT W0.00  ; 手/自动切换HMI
AND T0058  ; 上料提升气缸缩回位延时
AND T0010  ; 右升降缸原位延时
AND T0014  ; 上料左升降气缸缩回位时间
ANDNOT A280.04  ; 上料机械手脉冲输出中
ANDNOT W15.11  ; 上料机械手手动到腔体2位置
AND H53.00  ; 上料轴归零完成
AND W9.15  ; 上料机械手回#2腔体安全条件
@AND W3.05  ; 腔体2位置-HMI
LD W15.11  ; 上料机械手手动到腔体2位置
AND W9.02  ; 上料机械手在腔体2位置
OR W400.00  ; 总复位信号
KEEP(011) W15.11  ; 上料机械手手动到腔体2位置
; rung 10
LDNOT W0.00  ; 手/自动切换HMI
AND T0058  ; 上料提升气缸缩回位延时
AND T0010  ; 右升降缸原位延时
AND T0014  ; 上料左升降气缸缩回位时间
ANDNOT A280.04  ; 上料机械手脉冲输出中
ANDNOT W15.11  ; 上料机械手手动到腔体2位置
AND H53.00  ; 上料轴归零完成
AND W10.00  ; 上料机械手回NG槽安全条件
@AND W7.02  ; 扫码左NG HMI
AND<=F(332) D196 D30  ; 下料机械手当前位置(mm), 下料机械手NG放料位置(mm)
LD W15.00  ; 上料扫码左NG槽手动
AND W91.01  ; 上料机械手在右NG槽位置
OR W400.00  ; 总复位信号
KEEP(011) W15.00  ; 上料扫码左NG槽手动
; rung 11
LDNOT W0.00  ; 手/自动切换HMI
AND T0058  ; 上料提升气缸缩回位延时
AND T0010  ; 右升降缸原位延时
AND T0014  ; 上料左升降气缸缩回位时间
ANDNOT A280.04  ; 上料机械手脉冲输出中
ANDNOT W15.11  ; 上料机械手手动到腔体2位置
AND H53.00  ; 上料轴归零完成
AND W10.00  ; 上料机械手回NG槽安全条件
@AND W7.03  ; 扫码右NG HMI
AND<=F(332) D196 D30  ; 下料机械手当前位置(mm), 下料机械手NG放料位置(mm)
LD W15.01  ; 上料扫码右NG槽手动
AND W91.00  ; 上料机械手在左NG槽位置
OR W400.00  ; 总复位信号
KEEP(011) W15.01  ; 上料扫码右NG槽手动
; rung 12
LD W15.11  ; 上料机械手手动到腔体2位置
AND P_Off
OUT W3.05  ; 腔体2位置-HMI

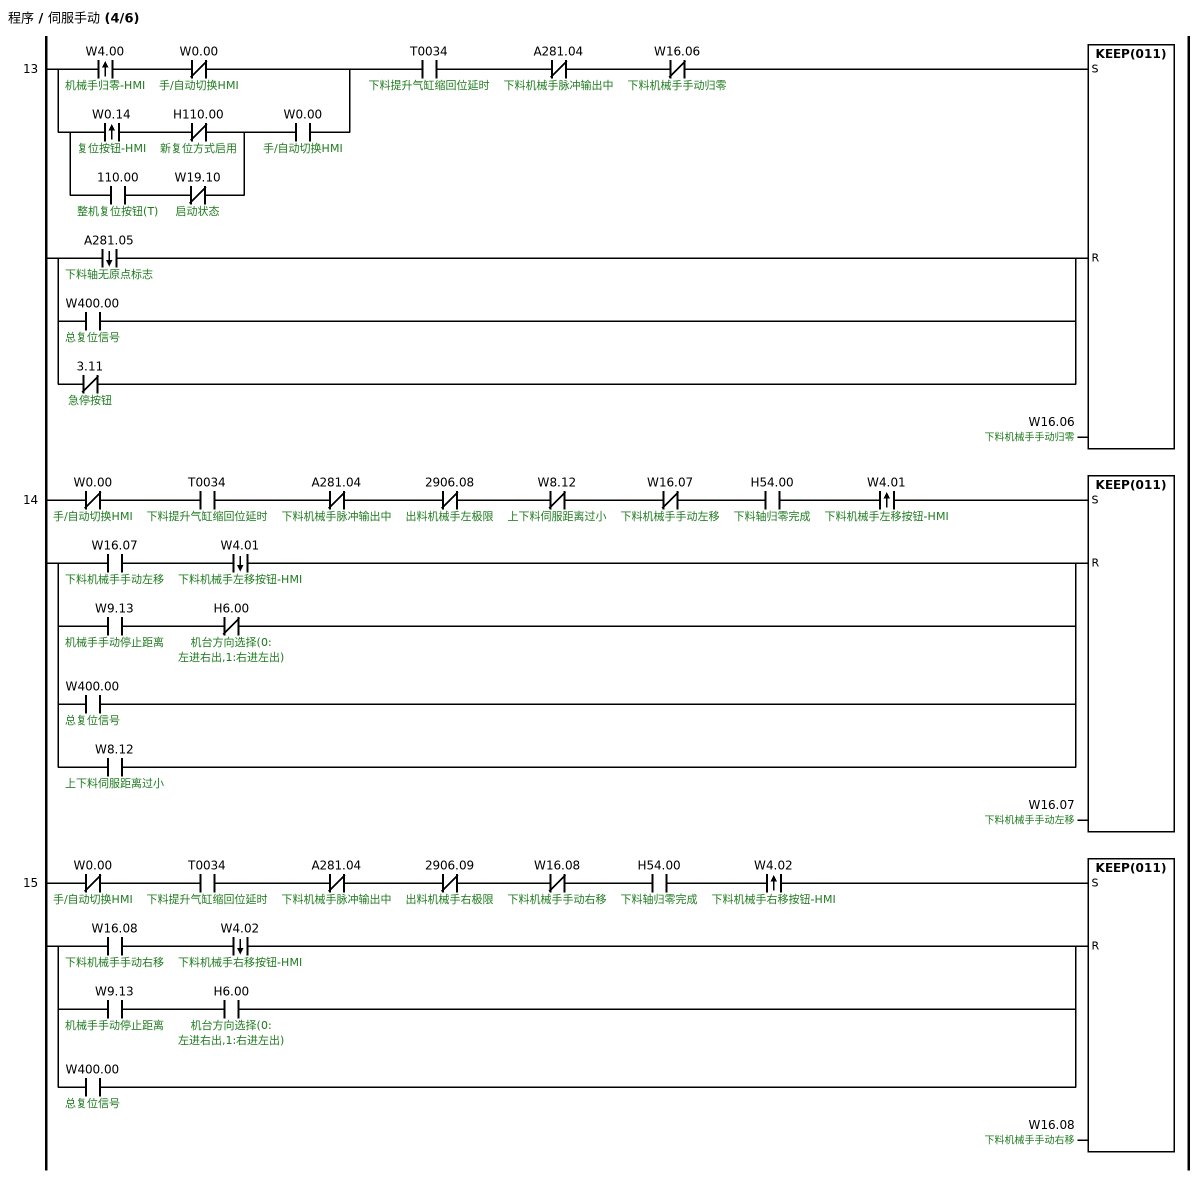
; rung 13
@LD W4.00  ; 机械手归零-HMI
ANDNOT W0.00  ; 手/自动切换HMI
@LD W0.14  ; 复位按钮-HMI
ANDNOT H110.00  ; 新复位方式启用
LD 110.00  ; 整机复位按钮(T)
ANDNOT W19.10  ; 启动状态
ORLD
AND W0.00  ; 手/自动切换HMI
ORLD
AND T0034  ; 下料提升气缸缩回位延时
ANDNOT A281.04  ; 下料机械手脉冲输出中
ANDNOT W16.06  ; 下料机械手手动归零
%LD A281.05  ; 下料轴无原点标志
OR W400.00  ; 总复位信号
ORNOT 3.11  ; 急停按钮
KEEP(011) W16.06  ; 下料机械手手动归零
; rung 14
LDNOT W0.00  ; 手/自动切换HMI
AND T0034  ; 下料提升气缸缩回位延时
ANDNOT A281.04  ; 下料机械手脉冲输出中
ANDNOT 2906.08  ; 出料机械手左极限
ANDNOT W8.12  ; 上下料伺服距离过小
ANDNOT W16.07  ; 下料机械手手动左移
AND H54.00  ; 下料轴归零完成
@AND W4.01  ; 下料机械手左移按钮-HMI
LD W16.07  ; 下料机械手手动左移
%AND W4.01  ; 下料机械手左移按钮-HMI
LD W9.13  ; 机械手手动停止距离
ANDNOT H6.00  ; 机台方向选择(0:左进右出,1:右进左出)
ORLD
OR W400.00  ; 总复位信号
OR W8.12  ; 上下料伺服距离过小
KEEP(011) W16.07  ; 下料机械手手动左移
; rung 15
LDNOT W0.00  ; 手/自动切换HMI
AND T0034  ; 下料提升气缸缩回位延时
ANDNOT A281.04  ; 下料机械手脉冲输出中
ANDNOT 2906.09  ; 出料机械手右极限
ANDNOT W16.08  ; 下料机械手手动右移
AND H54.00  ; 下料轴归零完成
@AND W4.02  ; 下料机械手右移按钮-HMI
LD W16.08  ; 下料机械手手动右移
%AND W4.02  ; 下料机械手右移按钮-HMI
LD W9.13  ; 机械手手动停止距离
AND H6.00  ; 机台方向选择(0:左进右出,1:右进左出)
ORLD
OR W400.00  ; 总复位信号
KEEP(011) W16.08  ; 下料机械手手动右移

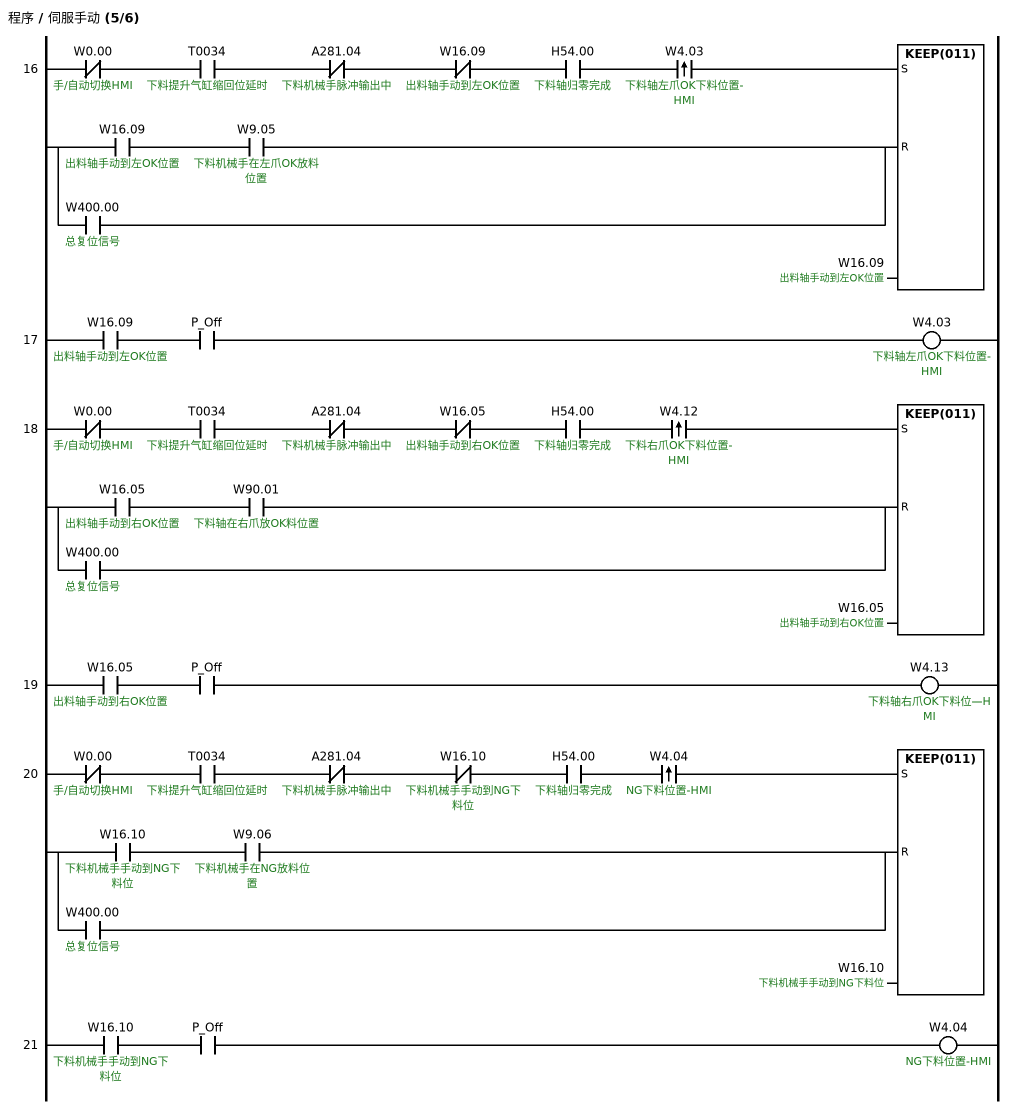
; rung 16
LDNOT W0.00  ; 手/自动切换HMI
AND T0034  ; 下料提升气缸缩回位延时
ANDNOT A281.04  ; 下料机械手脉冲输出中
ANDNOT W16.09  ; 出料轴手动到左OK位置
AND H54.00  ; 下料轴归零完成
@AND W4.03  ; 下料轴左爪OK下料位置-HMI
LD W16.09  ; 出料轴手动到左OK位置
AND W9.05  ; 下料机械手在左爪OK放料位置
OR W400.00  ; 总复位信号
KEEP(011) W16.09  ; 出料轴手动到左OK位置
; rung 17
LD W16.09  ; 出料轴手动到左OK位置
AND P_Off
OUT W4.03  ; 下料轴左爪OK下料位置-HMI
; rung 18
LDNOT W0.00  ; 手/自动切换HMI
AND T0034  ; 下料提升气缸缩回位延时
ANDNOT A281.04  ; 下料机械手脉冲输出中
ANDNOT W16.05  ; 出料轴手动到右OK位置
AND H54.00  ; 下料轴归零完成
@AND W4.12  ; 下料右爪OK下料位置-HMI
LD W16.05  ; 出料轴手动到右OK位置
AND W90.01  ; 下料轴在右爪放OK料位置
OR W400.00  ; 总复位信号
KEEP(011) W16.05  ; 出料轴手动到右OK位置
; rung 19
LD W16.05  ; 出料轴手动到右OK位置
AND P_Off
OUT W4.13  ; 下料轴右爪OK下料位—HMI
; rung 20
LDNOT W0.00  ; 手/自动切换HMI
AND T0034  ; 下料提升气缸缩回位延时
ANDNOT A281.04  ; 下料机械手脉冲输出中
ANDNOT W16.10  ; 下料机械手手动到NG下料位
AND H54.00  ; 下料轴归零完成
@AND W4.04  ; NG下料位置-HMI
LD W16.10  ; 下料机械手手动到NG下料位
AND W9.06  ; 下料机械手在NG放料位置
OR W400.00  ; 总复位信号
KEEP(011) W16.10  ; 下料机械手手动到NG下料位
; rung 21
LD W16.10  ; 下料机械手手动到NG下料位
AND P_Off
OUT W4.04  ; NG下料位置-HMI

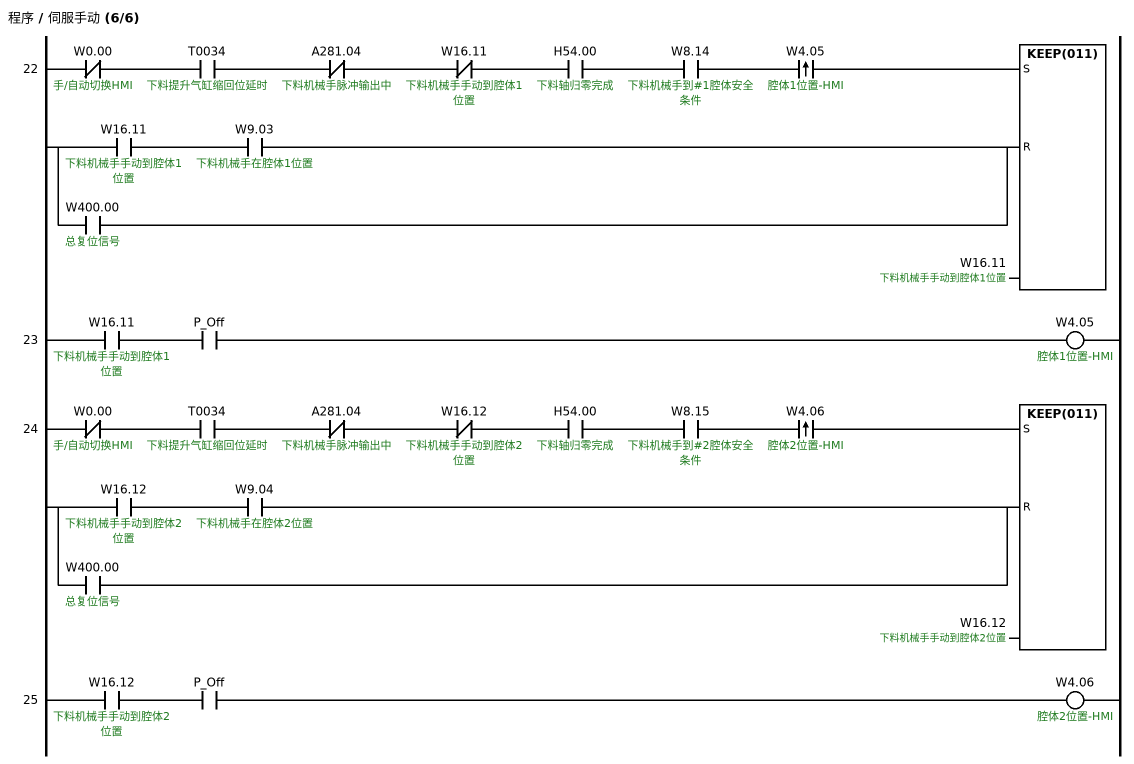
; rung 22
LDNOT W0.00  ; 手/自动切换HMI
AND T0034  ; 下料提升气缸缩回位延时
ANDNOT A281.04  ; 下料机械手脉冲输出中
ANDNOT W16.11  ; 下料机械手手动到腔体1位置
AND H54.00  ; 下料轴归零完成
AND W8.14  ; 下料机械手到#1腔体安全条件
@AND W4.05  ; 腔体1位置-HMI
LD W16.11  ; 下料机械手手动到腔体1位置
AND W9.03  ; 下料机械手在腔体1位置
OR W400.00  ; 总复位信号
KEEP(011) W16.11  ; 下料机械手手动到腔体1位置
; rung 23
LD W16.11  ; 下料机械手手动到腔体1位置
AND P_Off
OUT W4.05  ; 腔体1位置-HMI
; rung 24
LDNOT W0.00  ; 手/自动切换HMI
AND T0034  ; 下料提升气缸缩回位延时
ANDNOT A281.04  ; 下料机械手脉冲输出中
ANDNOT W16.12  ; 下料机械手手动到腔体2位置
AND H54.00  ; 下料轴归零完成
AND W8.15  ; 下料机械手到#2腔体安全条件
@AND W4.06  ; 腔体2位置-HMI
LD W16.12  ; 下料机械手手动到腔体2位置
AND W9.04  ; 下料机械手在腔体2位置
OR W400.00  ; 总复位信号
KEEP(011) W16.12  ; 下料机械手手动到腔体2位置
; rung 25
LD W16.12  ; 下料机械手手动到腔体2位置
AND P_Off
OUT W4.06  ; 腔体2位置-HMI

### Section 轴输出

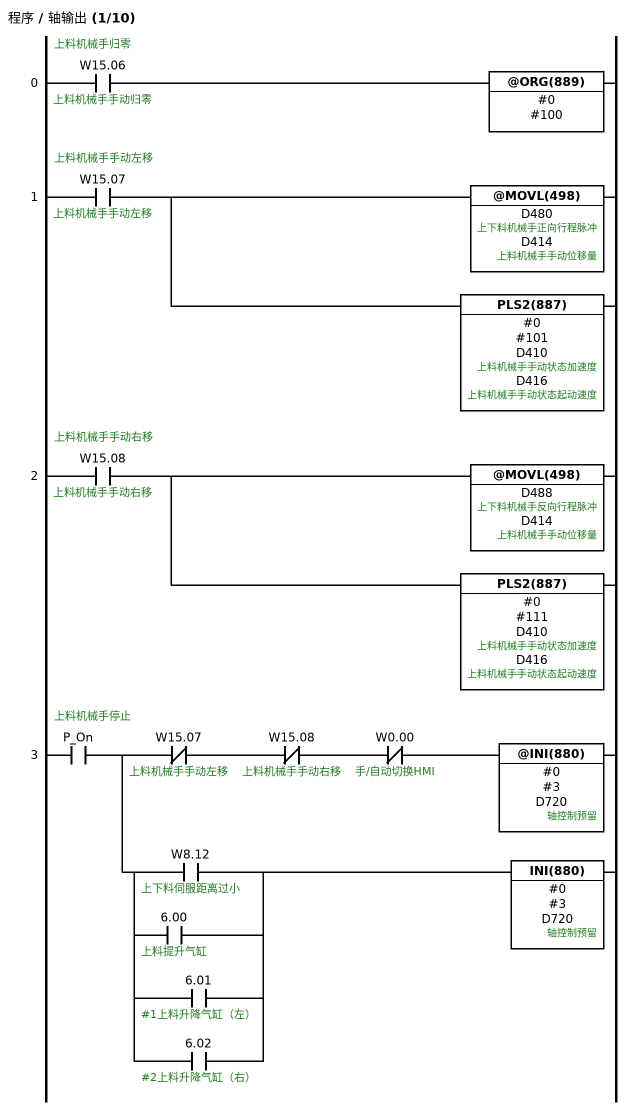
; rung 0: 上料机械手归零
LD W15.06  ; 上料机械手手动归零
@ORG(889) #0 #100
; rung 1: 上料机械手手动左移
LD W15.07  ; 上料机械手手动左移
@MOVL(498) D480 D414  ; 上下料机械手正向行程脉冲, 上料机械手手动位移量
PLS2(887) #0 #101 D410 D416  ; 上料机械手手动状态加速度, 上料机械手手动状态起动速度
; rung 2: 上料机械手手动右移
LD W15.08  ; 上料机械手手动右移
@MOVL(498) D488 D414  ; 上下料机械手反向行程脉冲, 上料机械手手动位移量
PLS2(887) #0 #111 D410 D416  ; 上料机械手手动状态加速度, 上料机械手手动状态起动速度
; rung 3: 上料机械手停止
LD P_On
OUT TR0
ANDNOT W15.07  ; 上料机械手手动左移
ANDNOT W15.08  ; 上料机械手手动右移
ANDNOT W0.00  ; 手/自动切换HMI
@INI(880) #0 #3 D720  ; 轴控制预留
LD TR0
LD W8.12  ; 上下料伺服距离过小
OR 6.00  ; 上料提升气缸
OR 6.01  ; #1上料升降气缸（左）
OR 6.02  ; #2上料升降气缸（右）
ANDLD
INI(880) #0 #3 D720  ; 轴控制预留

